C07281=1116.818,241.183,-70.393,-178.585,9.836,149.565
C07282=1116.821,240.934,-70.365,-178.587,9.834,149.565
C07283=1116.826,240.686,-70.337,-178.590,9.831,149.565
C07284=1116.829,240.473,-70.314,-178.593,9.829,149.565
C07285=1116.833,240.259,-70.290,-178.594,9.827,149.565
C07286=1116.837,240.046,-70.266,-178.597,9.825,149.565
C07287=1116.841,239.833,-70.242,-178.599,9.822,149.565
C07288=1116.844,239.620,-70.219,-178.601,9.820,149.565
C07289=1116.848,239.406,-70.195,-178.603,9.818,149.565
C07290=1116.851,239.193,-70.171,-178.605,9.816,149.565
C07291=1116.856,238.980,-70.147,-178.608,9.814,149.565
C07292=1116.860,238.732,-70.119,-178.610,9.811,149.565
C07293=1116.864,238.483,-70.092,-178.612,9.809,149.566
C07294=1116.869,238.235,-70.064,-178.615,9.806,149.566
C07295=1116.873,237.987,-70.036,-178.618,9.804,149.566
C07296=1116.877,237.738,-70.009,-178.620,9.801,149.566
C07297=1116.881,237.490,-69.981,-178.623,9.799,149.566
C07298=1116.886,237.242,-69.954,-178.626,9.796,149.566
C07299=1116.890,236.992,-69.927,-178.628,9.794,149.566
C07300=1116.894,236.744,-69.899,-178.631,9.791,149.566
C07301=1116.899,236.496,-69.872,-178.634,9.788,149.566
C07302=1116.903,236.247,-69.844,-178.637,9.785,149.566
C07303=1116.907,235.999,-69.817,-178.639,9.783,149.566
C07304=1116.912,235.751,-69.789,-178.642,9.780,149.567
C07305=1116.916,235.502,-69.761,-178.645,9.778,149.567
C07306=1116.921,235.253,-69.734,-178.648,9.775,149.567
C07307=1116.925,235.005,-69.707,-178.650,9.772,149.567
C07308=1116.930,234.757,-69.680,-178.653,9.769,149.567
C07309=1116.934,234.508,-69.652,-178.656,9.766,149.567
C07310=1116.938,234.260,-69.624,-178.659,9.764,149.567
C07311=1116.943,234.011,-69.597,-178.662,9.761,149.567
C07312=1116.946,233.762,-69.570,-178.665,9.758,149.567
C07313=1116.950,233.515,-69.543,-178.668,9.755,149.567
C07314=1116.955,233.266,-69.516,-178.671,9.753,149.568
C07315=1116.960,233.018,-69.489,-178.674,9.750,149.567
C07316=1116.964,232.768,-69.461,-178.677,9.747,149.568
C07317=1116.968,232.521,-69.433,-178.680,9.744,149.568
C07318=1116.973,232.272,-69.406,-178.682,9.741,149.568
C07319=1116.977,232.024,-69.379,-178.685,9.739,149.568
C07320=1116.981,231.775,-69.353,-178.688,9.736,149.568
C07321=1116.985,231.526,-69.325,-178.691,9.733,149.568
C07322=1116.990,231.278,-69.298,-178.694,9.730,149.568
C07323=1116.994,231.030,-69.270,-178.697,9.726,149.568
C07324=1116.999,230.781,-69.243,-178.700,9.724,149.568
C07325=1117.003,230.533,-69.217,-178.703,9.721,149.569
C07326=1117.007,230.284,-69.189,-178.706,9.718,149.569
C07327=1117.012,230.035,-69.162,-178.709,9.714,149.569
C07328=1117.016,229.787,-69.135,-178.712,9.712,149.569
C07329=1117.021,229.538,-69.108,-178.716,9.708,149.569
C07330=1117.025,229.290,-69.082,-178.719,9.705,149.569
C07331=1117.029,229.042,-69.055,-178.721,9.702,149.569
C07332=1117.034,228.793,-69.028,-178.725,9.699,149.569
C07333=1117.038,228.544,-69.000,-178.728,9.696,149.569
C07334=1117.042,228.296,-68.974,-178.730,9.693,149.569
C07335=1117.047,228.047,-68.947,-178.734,9.689,149.569
C07336=1117.051,227.799,-68.920,-178.737,9.686,149.569
C07337=1117.055,227.551,-68.893,-178.739,9.683,149.569
C07338=1117.060,227.302,-68.866,-178.742,9.681,149.569
C07339=1117.065,227.054,-68.839,-178.746,9.677,149.569
C07340=1117.068,226.840,-68.817,-178.747,9.674,149.569
C07341=1117.072,226.627,-68.793,-178.750,9.672,149.569
C07342=1117.076,226.414,-68.771,-178.753,9.669,149.569
C07343=1117.079,226.201,-68.747,-178.755,9.666,149.569
C07344=1117.083,225.987,-68.724,-178.758,9.663,149.569
C07345=1117.087,225.774,-68.702,-178.760,9.661,149.569
C07346=1117.090,225.561,-68.679,-178.762,9.658,149.569
C07347=1117.095,225.347,-68.656,-178.765,9.655,149.569
C07348=1117.099,225.099,-68.629,-178.768,9.652,149.569
C07349=1117.103,224.850,-68.602,-178.770,9.649,149.569
C07350=1117.107,224.601,-68.575,-178.773,9.646,149.569
C07351=1117.111,224.352,-68.549,-178.775,9.643,149.569
C07352=1117.116,224.104,-68.522,-178.778,9.640,149.569
C07353=1117.120,223.856,-68.496,-178.781,9.636,149.569
C07354=1117.125,223.607,-68.469,-178.784,9.633,149.569
C07355=1117.129,223.358,-68.443,-178.786,9.630,149.569
C07356=1117.134,223.110,-68.416,-178.789,9.627,149.569
C07357=1117.138,222.861,-68.389,-178.792,9.624,149.569
C07358=1117.142,222.613,-68.363,-178.794,9.621,149.569
C07359=1117.146,222.364,-68.336,-178.797,9.618,149.569
C07360=1117.151,222.115,-68.310,-178.799,9.614,149.569
C07361=1117.155,221.867,-68.284,-178.802,9.611,149.569
C07362=1117.160,221.619,-68.257,-178.804,9.608,149.569
C07363=1117.164,221.370,-68.231,-178.807,9.605,149.568
C07364=1117.169,221.121,-68.204,-178.809,9.602,149.568
C07365=1117.174,220.873,-68.178,-178.812,9.599,149.568
C07366=1117.178,220.625,-68.151,-178.814,9.595,149.568
C07367=1117.182,220.376,-68.126,-178.816,9.592,149.568
C07368=1117.187,220.127,-68.099,-178.819,9.589,149.568
C07369=1117.191,219.879,-68.072,-178.821,9.586,149.568
C07370=1117.195,219.630,-68.046,-178.824,9.583,149.568
C07371=1117.200,219.382,-68.019,-178.826,9.581,149.568
C07372=1117.204,219.133,-67.993,-178.828,9.577,149.568
C07373=1117.208,218.884,-67.968,-178.830,9.574,149.567
C07374=1117.213,218.636,-67.941,-178.833,9.571,149.567
C07375=1117.217,218.387,-67.915,-178.835,9.568,149.567
C07376=1117.222,218.139,-67.888,-178.837,9.566,149.567
C07377=1117.226,217.890,-67.862,-178.839,9.562,149.567
C07378=1117.230,217.642,-67.836,-178.842,9.559,149.567
C07379=1117.236,217.393,-67.810,-178.845,9.556,149.567
C07380=1117.240,217.144,-67.784,-178.846,9.553,149.567
C07381=1117.244,216.896,-67.757,-178.849,9.550,149.567
C07382=1117.248,216.647,-67.732,-178.851,9.547,149.566
C07383=1117.253,216.398,-67.705,-178.854,9.544,149.566
C07384=1117.257,216.150,-67.679,-178.855,9.541,149.566
C07385=1117.261,215.901,-67.653,-178.858,9.538,149.566
C07386=1117.266,215.652,-67.627,-178.859,9.536,149.566
C07387=1117.271,215.405,-67.601,-178.862,9.533,149.566
C07388=1117.275,215.156,-67.575,-178.864,9.529,149.566
C07389=1117.279,214.907,-67.549,-178.866,9.527,149.566
C07390=1117.284,214.659,-67.522,-178.869,9.524,149.566
C07391=1117.288,214.410,-67.496,-178.870,9.521,149.565
C07392=1117.292,214.161,-67.471,-178.873,9.518,149.565
C07393=1117.297,213.913,-67.445,-178.874,9.515,149.565
C07394=1117.301,213.665,-67.419,-178.877,9.512,149.565
C07395=1117.306,213.416,-67.392,-178.878,9.510,149.565
C07396=1117.309,213.202,-67.370,-178.881,9.507,149.565
C07397=1117.313,212.988,-67.349,-178.883,9.504,149.565
C07398=1117.317,212.775,-67.326,-178.885,9.502,149.565
C07399=1117.321,212.562,-67.304,-178.887,9.499,149.565
C07400=1117.325,212.348,-67.281,-178.889,9.496,149.565
C07401=1117.328,212.135,-67.259,-178.891,9.494,149.565
C07402=1117.332,211.921,-67.237,-178.894,9.491,149.565
C07403=1117.336,211.707,-67.215,-178.896,9.489,149.565
C07404=1117.340,211.459,-67.189,-178.898,9.486,149.565
C07405=1117.345,211.210,-67.164,-178.901,9.483,149.565
C07406=1117.349,210.962,-67.138,-178.903,9.480,149.565
C07407=1117.354,210.713,-67.112,-178.906,9.478,149.565
C07408=1117.359,210.464,-67.086,-178.908,9.475,149.565
C07409=1117.363,210.216,-67.061,-178.911,9.472,149.565
C07410=1117.367,209.967,-67.034,-178.914,9.469,149.565
C07411=1117.371,209.719,-67.008,-178.916,9.466,149.565
C07412=1117.376,209.471,-66.983,-178.919,9.463,149.565
C07413=1117.380,209.222,-66.957,-178.922,9.460,149.565
C07414=1117.385,208.972,-66.932,-178.925,9.457,149.565
C07415=1117.389,208.724,-66.907,-178.927,9.454,149.565
C07416=1117.394,208.475,-66.881,-178.930,9.451,149.565
C07417=1117.398,208.227,-66.855,-178.933,9.448,149.565
C07418=1117.402,207.978,-66.829,-178.936,9.445,149.565
C07419=1117.407,207.730,-66.804,-178.939,9.443,149.565
C07420=1117.411,207.481,-66.778,-178.941,9.440,149.565
C07421=1117.415,207.232,-66.753,-178.944,9.437,149.565
C07422=1117.420,206.984,-66.727,-178.947,9.434,149.565
C07423=1117.424,206.735,-66.701,-178.950,9.431,149.565
C07424=1117.429,206.486,-66.676,-178.953,9.428,149.566
C07425=1117.434,206.238,-66.651,-178.955,9.425,149.566
C07426=1117.438,205.989,-66.625,-178.958,9.422,149.566
C07427=1117.443,205.741,-66.600,-178.961,9.420,149.566
C07428=1117.447,205.492,-66.574,-178.964,9.417,149.566
C07429=1117.452,205.242,-66.549,-178.967,9.414,149.566
C07430=1117.456,204.994,-66.524,-178.969,9.411,149.566
C07431=1117.461,204.746,-66.498,-178.972,9.408,149.566
C07432=1117.465,204.497,-66.472,-178.975,9.406,149.566
C07433=1117.470,204.248,-66.448,-178.978,9.403,149.566
C07434=1117.474,203.999,-66.422,-178.981,9.400,149.566
C07435=1117.478,203.751,-66.397,-178.984,9.397,149.567
C07436=1117.483,203.503,-66.371,-178.987,9.394,149.567
C07437=1117.487,203.253,-66.346,-178.990,9.391,149.567
C07438=1117.492,203.005,-66.321,-178.993,9.388,149.567
C07439=1117.496,202.756,-66.296,-178.996,9.385,149.567
C07440=1117.501,202.508,-66.270,-178.999,9.382,149.567
C07441=1117.505,202.259,-66.245,-179.002,9.379,149.567
C07442=1117.510,202.010,-66.221,-179.004,9.376,149.567
C07443=1117.514,201.762,-66.195,-179.008,9.373,149.567
C07444=1117.519,201.512,-66.170,-179.011,9.370,149.567
C07445=1117.524,201.264,-66.144,-179.014,9.367,149.568
C07446=1117.527,201.016,-66.119,-179.016,9.364,149.568
C07447=1117.532,200.767,-66.095,-179.020,9.361,149.568
C07448=1117.536,200.518,-66.069,-179.023,9.358,149.568
C07449=1117.541,200.270,-66.045,-179.026,9.355,149.568
C07450=1117.545,200.021,-66.019,-179.028,9.352,149.568
C07451=1117.550,199.772,-65.994,-179.032,9.348,149.568
C07452=1117.554,199.558,-65.973,-179.034,9.345,149.568
C07453=1117.558,199.345,-65.952,-179.037,9.343,149.568
C07454=1117.562,199.131,-65.930,-179.040,9.341,149.568
C07455=1117.565,198.918,-65.908,-179.042,9.338,149.568
C07456=1117.569,198.704,-65.887,-179.045,9.335,149.568
C07457=1117.573,198.490,-65.866,-179.047,9.332,149.568
C07458=1117.577,198.277,-65.844,-179.050,9.330,149.568
C07459=1117.580,198.063,-65.823,-179.052,9.327,149.568
C07460=1117.586,197.814,-65.798,-179.056,9.323,149.569
C07461=1117.589,197.566,-65.773,-179.058,9.320,149.569
C07462=1117.594,197.317,-65.748,-179.062,9.317,149.569
C07463=1117.599,197.068,-65.723,-179.065,9.313,149.569
C07464=1117.603,196.820,-65.699,-179.068,9.310,149.569
C07465=1117.607,196.571,-65.674,-179.071,9.307,149.569
C07466=1117.612,196.322,-65.649,-179.074,9.303,149.569
C07467=1117.617,196.073,-65.625,-179.076,9.301,149.569
C07468=1117.620,195.825,-65.600,-179.077,9.298,149.568
C07469=1117.626,195.576,-65.575,-179.080,9.295,149.568
C07470=1117.630,195.327,-65.550,-179.081,9.292,149.568
C07471=1117.634,195.078,-65.526,-179.083,9.290,149.568
C07472=1117.640,194.830,-65.501,-179.085,9.287,149.568
C07473=1117.643,194.581,-65.476,-179.087,9.284,149.568
C07474=1117.648,194.332,-65.451,-179.089,9.282,149.568
C07475=1117.652,194.083,-65.427,-179.090,9.279,149.567
C07476=1117.657,193.835,-65.402,-179.093,9.276,149.567
C07477=1117.661,193.586,-65.378,-179.095,9.273,149.567
C07478=1117.666,193.337,-65.353,-179.097,9.270,149.567
C07479=1117.670,193.088,-65.329,-179.099,9.268,149.567
C07480=1117.675,192.840,-65.304,-179.101,9.265,149.567
C07481=1117.679,192.591,-65.279,-179.103,9.262,149.567
C07482=1117.684,192.342,-65.255,-179.105,9.260,149.567
C07483=1117.689,192.094,-65.231,-179.108,9.257,149.567
C07484=1117.693,191.845,-65.205,-179.109,9.254,149.567
C07485=1117.697,191.596,-65.181,-179.111,9.252,149.567
C07486=1117.703,191.347,-65.157,-179.114,9.249,149.567
C07487=1117.706,191.098,-65.132,-179.115,9.246,149.567
C07488=1117.711,190.850,-65.108,-179.118,9.243,149.567
C07489=1117.716,190.601,-65.084,-179.120,9.241,149.566
C07490=1117.720,190.352,-65.059,-179.122,9.238,149.566
C07491=1117.725,190.103,-65.034,-179.124,9.235,149.566
C07492=1117.729,189.855,-65.010,-179.127,9.232,149.566
C07493=1117.733,189.606,-64.986,-179.129,9.230,149.566
C07494=1117.738,189.357,-64.961,-179.131,9.226,149.566
C07495=1117.743,189.109,-64.937,-179.133,9.223,149.566
C07496=1117.748,188.860,-64.913,-179.135,9.221,149.566
C07497=1117.752,188.611,-64.888,-179.138,9.218,149.566
C07498=1117.756,188.362,-64.865,-179.140,9.216,149.566
C07499=1117.761,188.113,-64.840,-179.143,9.213,149.566
C07500=1117.766,187.865,-64.816,-179.145,9.210,149.566
C07501=1117.770,187.616,-64.792,-179.147,9.207,149.566
C07502=1117.775,187.367,-64.767,-179.150,9.204,149.566
C07503=1117.779,187.118,-64.743,-179.152,9.201,149.566
C07504=1117.783,186.870,-64.719,-179.154,9.199,149.566
C07505=1117.788,186.620,-64.694,-179.156,9.196,149.566
C07506=1117.793,186.372,-64.670,-179.159,9.193,149.566
C07507=1117.797,186.123,-64.646,-179.161,9.190,149.566
C07508=1117.801,185.910,-64.625,-179.163,9.187,149.566
C07509=1117.805,185.695,-64.604,-179.165,9.185,149.566
C07510=1117.809,185.482,-64.584,-179.167,9.183,149.566
C07511=1117.813,185.268,-64.563,-179.169,9.180,149.566
C07512=1117.817,185.055,-64.542,-179.172,9.177,149.566
C07513=1117.821,184.841,-64.522,-179.174,9.175,149.565
C07514=1117.824,184.627,-64.501,-179.176,9.173,149.566
C07515=1117.829,184.413,-64.480,-179.178,9.170,149.566
C07516=1117.833,184.165,-64.456,-179.180,9.167,149.566
C07517=1117.837,183.916,-64.432,-179.183,9.164,149.566
C07518=1117.842,183.667,-64.408,-179.185,9.161,149.565
C07519=1117.846,183.418,-64.384,-179.188,9.158,149.565
C07520=1117.850,183.170,-64.360,-179.190,9.155,149.565
C07521=1117.856,182.920,-64.336,-179.193,9.152,149.565
C07522=1117.860,182.672,-64.312,-179.195,9.149,149.565
C07523=1117.865,182.424,-64.288,-179.198,9.146,149.565
C07524=1117.869,182.175,-64.265,-179.201,9.143,149.565
C07525=1117.873,181.926,-64.240,-179.203,9.140,149.565
C07526=1117.878,181.676,-64.217,-179.206,9.137,149.565
C07527=1117.882,181.428,-64.193,-179.208,9.134,149.565
C07528=1117.888,181.179,-64.169,-179.211,9.130,149.565
C07529=1117.892,180.930,-64.145,-179.214,9.127,149.565
C07530=1117.897,180.681,-64.122,-179.216,9.124,149.565
C07531=1117.901,180.433,-64.097,-179.219,9.121,149.565
C07532=1117.906,180.184,-64.074,-179.221,9.118,149.565
C07533=1117.910,179.935,-64.050,-179.224,9.114,149.565
C07534=1117.914,179.686,-64.026,-179.227,9.111,149.565
C07535=1117.919,179.437,-64.002,-179.229,9.108,149.565
C07536=1117.923,179.188,-63.979,-179.232,9.105,149.565
C07537=1117.928,178.940,-63.955,-179.234,9.102,149.565
C07538=1117.932,178.691,-63.931,-179.236,9.099,149.565
C07539=1117.937,178.442,-63.908,-179.238,9.096,149.565
C07540=1117.942,178.193,-63.884,-179.240,9.094,149.565
C07541=1117.946,177.944,-63.861,-179.242,9.090,149.564
C07542=1117.951,177.696,-63.837,-179.245,9.087,149.564
C07543=1117.955,177.447,-63.813,-179.247,9.085,149.564
C07544=1117.960,177.198,-63.790,-179.249,9.081,149.564
C07545=1117.964,176.949,-63.766,-179.251,9.078,149.564
C07546=1117.969,176.700,-63.742,-179.253,9.076,149.564
C07547=1117.974,176.451,-63.719,-179.256,9.073,149.564
C07548=1117.979,176.202,-63.696,-179.258,9.069,149.564
C07549=1117.983,175.954,-63.672,-179.260,9.067,149.564
C07550=1117.988,175.705,-63.648,-179.262,9.064,149.564
C07551=1117.992,175.456,-63.625,-179.264,9.060,149.563
C07552=1117.997,175.207,-63.601,-179.266,9.058,149.563
C07553=1118.001,174.959,-63.578,-179.269,9.055,149.563
C07554=1118.005,174.710,-63.555,-179.271,9.051,149.563
C07555=1118.010,174.461,-63.531,-179.273,9.049,149.563
C07556=1118.015,174.212,-63.508,-179.275,9.046,149.563
C07557=1118.019,173.963,-63.484,-179.277,9.042,149.563
C07558=1118.024,173.714,-63.461,-179.279,9.040,149.563
C07559=1118.029,173.465,-63.437,-179.282,9.037,149.563
C07560=1118.033,173.216,-63.414,-179.284,9.033,149.562
C07561=1118.037,172.967,-63.391,-179.286,9.031,149.562
C07562=1118.042,172.718,-63.368,-179.288,9.028,149.562
C07563=1118.047,172.469,-63.344,-179.291,9.025,149.562
C07564=1118.050,172.256,-63.325,-179.292,9.022,149.562
C07565=1118.055,172.042,-63.304,-179.294,9.020,149.562
C07566=1118.058,171.828,-63.284,-179.296,9.017,149.562
C07567=1118.062,171.614,-63.264,-179.299,9.014,149.562
C07568=1118.066,171.400,-63.244,-179.300,9.012,149.562
C07569=1118.070,171.187,-63.224,-179.302,9.009,149.562
C07570=1118.074,170.973,-63.204,-179.304,9.007,149.562
C07571=1118.078,170.759,-63.184,-179.306,9.005,149.562
C07572=1118.082,170.510,-63.161,-179.308,9.001,149.561
C07573=1118.087,170.261,-63.138,-179.310,8.998,149.561
C07574=1118.092,170.012,-63.114,-179.313,8.995,149.561
C07575=1118.097,169.763,-63.091,-179.314,8.992,149.561
C07576=1118.101,169.515,-63.068,-179.317,8.989,149.561
C07577=1118.105,169.266,-63.045,-179.319,8.986,149.561
C07578=1118.111,169.017,-63.022,-179.321,8.983,149.561
C07579=1118.114,168.769,-62.999,-179.323,8.980,149.561
C07580=1118.119,168.520,-62.976,-179.326,8.977,149.561
C07581=1118.124,168.270,-62.952,-179.328,8.974,149.560
C07582=1118.129,168.021,-62.930,-179.330,8.971,149.560
C07583=1118.133,167.772,-62.907,-179.333,8.967,149.560
C07584=1118.138,167.523,-62.884,-179.334,8.965,149.560
C07585=1118.143,167.275,-62.861,-179.337,8.962,149.560
C07586=1118.147,167.026,-62.838,-179.339,8.958,149.560
C07587=1118.152,166.777,-62.814,-179.342,8.955,149.560
C07588=1118.156,166.528,-62.791,-179.344,8.952,149.560
C07589=1118.160,166.279,-62.769,-179.346,8.950,149.560
C07590=1118.166,166.030,-62.746,-179.348,8.946,149.559
C07591=1118.170,165.781,-62.723,-179.351,8.943,149.559
C07592=1118.174,165.533,-62.700,-179.353,8.940,149.559
C07593=1118.179,165.284,-62.677,-179.355,8.936,149.559
C07594=1118.183,165.034,-62.655,-179.358,8.933,149.559
C07595=1118.189,164.786,-62.632,-179.360,8.931,149.559
C07596=1118.193,164.537,-62.609,-179.362,8.927,149.559
C07597=1118.197,164.288,-62.585,-179.364,8.924,149.559
C07598=1118.202,164.038,-62.563,-179.367,8.921,149.559
C07599=1118.206,163.790,-62.540,-179.369,8.918,149.559
C07600=1118.212,163.541,-62.517,-179.371,8.915,149.559
C07601=1118.216,163.292,-62.495,-179.373,8.911,149.558
C07602=1118.221,163.043,-62.472,-179.376,8.908,149.558
C07603=1118.225,162.794,-62.449,-179.378,8.906,149.558
C07604=1118.230,162.545,-62.427,-179.380,8.902,149.558
C07605=1118.234,162.297,-62.404,-179.382,8.899,149.558
C07606=1118.239,162.047,-62.381,-179.385,8.896,149.558
C07607=1118.243,161.798,-62.358,-179.387,8.893,149.558
C07608=1118.248,161.550,-62.335,-179.390,8.889,149.558
C07609=1118.253,161.301,-62.313,-179.392,8.886,149.557
C07610=1118.257,161.052,-62.290,-179.394,8.883,149.557
C07611=1118.262,160.803,-62.268,-179.396,8.879,149.557
C07612=1118.266,160.554,-62.246,-179.399,8.876,149.557
C07613=1118.271,160.305,-62.223,-179.401,8.873,149.557
C07614=1118.276,160.057,-62.201,-179.403,8.870,149.557
C07615=1118.281,159.807,-62.178,-179.406,8.867,149.557
C07616=1118.285,159.558,-62.155,-179.408,8.863,149.557
C07617=1118.290,159.309,-62.133,-179.411,8.860,149.557
C07618=1118.294,159.060,-62.110,-179.413,8.856,149.556
C07619=1118.299,158.811,-62.088,-179.415,8.853,149.556
C07620=1118.304,158.551,-62.064,-179.417,8.850,149.556
C07621=1118.309,158.290,-62.041,-179.420,8.847,149.556
C07622=1118.314,158.030,-62.017,-179.422,8.843,149.556
C07623=1118.318,157.768,-61.994,-179.424,8.840,149.556
C07624=1118.323,157.520,-61.971,-179.426,8.837,149.555
C07625=1118.327,157.271,-61.949,-179.429,8.834,149.555
C07626=1118.332,157.023,-61.926,-179.431,8.830,149.555
C07627=1118.337,156.773,-61.904,-179.433,8.827,149.555
C07628=1118.341,156.524,-61.882,-179.436,8.823,149.555
C07629=1118.346,156.276,-61.860,-179.438,8.819,149.555
C07630=1118.351,156.026,-61.837,-179.441,8.816,149.555
C07631=1118.355,155.778,-61.815,-179.443,8.813,149.554
C07632=1118.360,155.528,-61.793,-179.445,8.810,149.554
C07633=1118.364,155.279,-61.770,-179.448,8.806,149.554
C07634=1118.369,155.031,-61.748,-179.450,8.803,149.554
C07635=1118.374,154.781,-61.726,-179.452,8.799,149.554
C07636=1118.378,154.533,-61.705,-179.454,8.796,149.554
C07637=1118.383,154.284,-61.681,-179.456,8.792,149.553
C07638=1118.388,154.035,-61.660,-179.459,8.789,149.553
C07639=1118.392,153.786,-61.638,-179.462,8.785,149.553
C07640=1118.397,153.536,-61.616,-179.464,8.782,149.553
C07641=1118.401,153.288,-61.594,-179.466,8.778,149.553
C07642=1118.406,153.038,-61.571,-179.468,8.775,149.553
C07643=1118.411,152.790,-61.549,-179.471,8.772,149.553
C07644=1118.415,152.541,-61.527,-179.473,8.768,149.552
C07645=1118.420,152.292,-61.505,-179.475,8.765,149.552
C07646=1118.424,152.043,-61.483,-179.478,8.761,149.552
C07647=1118.429,151.794,-61.461,-179.480,8.758,149.552
C07648=1118.434,151.544,-61.439,-179.482,8.754,149.552
C07649=1118.439,151.296,-61.417,-179.484,8.751,149.551
C07650=1118.443,151.046,-61.395,-179.486,8.747,149.551
C07651=1118.448,150.798,-61.373,-179.490,8.743,149.551
C07652=1118.453,150.548,-61.351,-179.492,8.740,149.551
C07653=1118.457,150.300,-61.330,-179.494,8.736,149.551
C07654=1118.462,150.051,-61.308,-179.496,8.733,149.550
C07655=1118.467,149.802,-61.286,-179.499,8.728,149.550
C07656=1118.471,149.553,-61.264,-179.501,8.725,149.550
C07657=1118.476,149.304,-61.242,-179.503,8.722,149.550
C07658=1118.481,149.055,-61.220,-179.505,8.718,149.550
C07659=1118.486,148.805,-61.198,-179.508,8.714,149.549
C07660=1118.490,148.557,-61.176,-179.510,8.711,149.549
C07661=1118.495,148.307,-61.154,-179.512,8.707,149.549
C07662=1118.500,148.059,-61.132,-179.514,8.704,149.549
C07663=1118.504,147.810,-61.111,-179.517,8.699,149.549
C07664=1118.509,147.560,-61.089,-179.519,8.696,149.548
C07665=1118.514,147.312,-61.068,-179.521,8.693,149.548
C07666=1118.518,147.062,-61.046,-179.524,8.689,149.548
C07667=1118.523,146.814,-61.024,-179.526,8.685,149.548
C07668=1118.530,146.397,-60.988,-179.530,8.679,149.547
C07669=1118.538,145.981,-60.952,-179.534,8.672,149.547
C07670=1118.546,145.565,-60.915,-179.538,8.666,149.547
C07671=1118.554,145.149,-60.880,-179.541,8.660,149.546
C07672=1118.558,144.935,-60.861,-179.543,8.657,149.546
C07673=1118.562,144.720,-60.843,-179.545,8.653,149.545
C07674=1118.566,144.506,-60.824,-179.546,8.651,149.545
C07675=1118.570,144.293,-60.805,-179.547,8.647,149.545
C07676=1118.574,144.078,-60.788,-179.548,8.645,149.545
C07677=1118.578,143.864,-60.768,-179.550,8.642,149.544
C07678=1118.582,143.651,-60.750,-179.551,8.639,149.544
C07679=1118.586,143.436,-60.732,-179.552,8.636,149.544
C07680=1118.591,143.187,-60.710,-179.554,8.633,149.543
C07681=1118.595,142.938,-60.689,-179.555,8.630,149.543
C07682=1118.600,142.689,-60.668,-179.558,8.626,149.543
C07683=1118.605,142.440,-60.646,-179.559,8.623,149.542
C07684=1118.609,142.191,-60.624,-179.561,8.620,149.542
C07685=1118.614,141.942,-60.603,-179.562,8.616,149.542
C07686=1118.618,141.694,-60.582,-179.564,8.613,149.541
C07687=1118.624,141.444,-60.561,-179.565,8.609,149.541
C07688=1118.628,141.195,-60.539,-179.567,8.606,149.541
C07689=1118.633,140.946,-60.518,-179.568,8.603,149.540
C07690=1118.638,140.697,-60.496,-179.570,8.599,149.540
C07691=1118.642,140.447,-60.476,-179.571,8.596,149.540
C07692=1118.647,140.199,-60.454,-179.574,8.592,149.539
C07693=1118.652,139.950,-60.432,-179.575,8.589,149.539
C07694=1118.657,139.701,-60.411,-179.577,8.586,149.539
C07695=1118.660,139.452,-60.390,-179.578,8.582,149.538
C07696=1118.665,139.203,-60.369,-179.580,8.579,149.538
C07697=1118.671,138.953,-60.348,-179.582,8.576,149.538
C07698=1118.675,138.705,-60.327,-179.583,8.573,149.537
C07699=1118.679,138.455,-60.306,-179.585,8.569,149.537
C07700=1118.684,138.206,-60.284,-179.587,8.565,149.537
C07701=1118.689,137.957,-60.263,-179.588,8.563,149.537
C07702=1118.693,137.709,-60.242,-179.590,8.559,149.536
C07703=1118.699,137.460,-60.221,-179.591,8.556,149.536
C07704=1118.703,137.210,-60.199,-179.593,8.553,149.536
C07705=1118.707,136.961,-60.178,-179.595,8.549,149.535
C07706=1118.713,136.712,-60.157,-179.596,8.546,149.535
C07707=1118.717,136.463,-60.136,-179.598,8.543,149.535
C07708=1118.722,136.214,-60.115,-179.599,8.539,149.534
C07709=1118.726,135.964,-60.094,-179.601,8.536,149.534
C07710=1118.731,135.716,-60.072,-179.603,8.532,149.534
C07711=1118.736,135.467,-60.052,-179.604,8.529,149.533
C07712=1118.741,135.218,-60.031,-179.607,8.526,149.533
C07713=1118.745,134.969,-60.011,-179.608,8.522,149.533
C07714=1118.750,134.720,-59.989,-179.610,8.519,149.533
C07715=1118.755,134.470,-59.968,-179.612,8.516,149.532
C07716=1118.759,134.221,-59.947,-179.613,8.513,149.532
C07717=1118.764,133.972,-59.926,-179.615,8.509,149.532
C07718=1118.769,133.724,-59.905,-179.617,8.506,149.531
C07719=1118.774,133.474,-59.884,-179.618,8.503,149.531
C07720=1118.779,133.225,-59.863,-179.620,8.499,149.531
C07721=1118.783,132.976,-59.843,-179.622,8.496,149.531
C07722=1118.788,132.727,-59.821,-179.623,8.493,149.530
C07723=1118.792,132.478,-59.800,-179.625,8.489,149.530
C07724=1118.797,132.228,-59.780,-179.626,8.486,149.530
C07725=1118.802,131.980,-59.759,-179.629,8.483,149.529
C07726=1118.807,131.730,-59.738,-179.630,8.479,149.529
C07727=1118.811,131.481,-59.718,-179.632,8.476,149.529
C07728=1118.815,131.267,-59.699,-179.633,8.474,149.529
C07729=1118.820,131.053,-59.681,-179.635,8.470,149.528
C07730=1118.823,130.839,-59.664,-179.637,8.467,149.528
C07731=1118.827,130.625,-59.646,-179.638,8.465,149.528
C07732=1118.831,130.411,-59.628,-179.639,8.462,149.528
C07733=1118.836,130.196,-59.610,-179.640,8.459,149.527
C07734=1118.839,129.983,-59.592,-179.642,8.456,149.527
C07735=1118.844,129.769,-59.574,-179.643,8.453,149.527
C07736=1118.849,129.520,-59.553,-179.645,8.450,149.527
C07737=1118.853,129.271,-59.533,-179.647,8.446,149.526
C07738=1118.858,129.022,-59.513,-179.648,8.443,149.526
C07739=1118.863,128.772,-59.492,-179.651,8.440,149.526
C07740=1118.867,128.523,-59.471,-179.653,8.436,149.525
C07741=1118.873,128.274,-59.450,-179.654,8.434,149.525
C07742=1118.877,128.025,-59.430,-179.656,8.430,149.525
C07743=1118.882,127.776,-59.409,-179.658,8.426,149.525
C07744=1118.887,127.527,-59.389,-179.659,8.423,149.524
C07745=1118.891,127.278,-59.368,-179.661,8.420,149.524
C07746=1118.896,127.029,-59.347,-179.663,8.416,149.524
C07747=1118.901,126.780,-59.327,-179.664,8.413,149.523
C07748=1118.905,126.531,-59.307,-179.666,8.410,149.523
C07749=1118.910,126.281,-59.285,-179.668,8.406,149.523
C07750=1118.914,126.031,-59.266,-179.669,8.403,149.523
C07751=1118.919,125.782,-59.245,-179.672,8.400,149.522
C07752=1118.925,125.534,-59.225,-179.674,8.396,149.522
C07753=1118.929,125.285,-59.204,-179.676,8.393,149.522
C07754=1118.933,125.036,-59.184,-179.677,8.390,149.522
C07755=1118.939,124.787,-59.163,-179.679,8.386,149.521
C07756=1118.943,124.538,-59.143,-179.681,8.383,149.521
C07757=1118.948,124.289,-59.122,-179.682,8.380,149.521
C07758=1118.953,124.039,-59.102,-179.684,8.377,149.521
C07759=1118.957,123.790,-59.082,-179.686,8.373,149.520
C07760=1118.962,123.541,-59.061,-179.687,8.370,149.520
C07761=1118.966,123.292,-59.041,-179.689,8.366,149.520
C07762=1118.972,123.042,-59.021,-179.692,8.363,149.519
C07763=1118.976,122.793,-59.000,-179.693,8.359,149.519
C07764=1118.981,122.544,-58.980,-179.695,8.356,149.519
C07765=1118.985,122.295,-58.959,-179.697,8.353,149.519
C07766=1118.991,122.045,-58.939,-179.699,8.349,149.518
C07767=1118.995,121.797,-58.919,-179.700,8.347,149.518
C07768=1118.999,121.548,-58.898,-179.702,8.343,149.518
C07769=1119.004,121.299,-58.878,-179.704,8.339,149.517
C07770=1119.009,121.050,-58.859,-179.706,8.336,149.517
C07771=1119.014,120.801,-58.838,-179.707,8.333,149.517
C07772=1119.019,120.552,-58.817,-179.709,8.329,149.517
C07773=1119.024,120.302,-58.798,-179.711,8.326,149.516
C07774=1119.028,120.053,-58.777,-179.713,8.322,149.516
C07775=1119.032,119.804,-58.757,-179.715,8.319,149.516
C07776=1119.037,119.555,-58.737,-179.717,8.316,149.516
C07777=1119.042,119.305,-58.716,-179.718,8.312,149.515
C07778=1119.048,119.056,-58.697,-179.720,8.309,149.515
C07779=1119.052,118.807,-58.677,-179.722,8.306,149.515
C07780=1119.057,118.558,-58.657,-179.724,8.302,149.515
C07781=1119.061,118.309,-58.637,-179.725,8.298,149.514
C07782=1119.066,118.060,-58.616,-179.727,8.295,149.514
C07783=1119.071,117.810,-58.597,-179.729,8.292,149.514
C07784=1119.075,117.597,-58.579,-179.731,8.289,149.513
C07785=1119.079,117.382,-58.563,-179.732,8.286,149.513
C07786=1119.083,117.168,-58.545,-179.734,8.283,149.513
C07787=1119.087,116.954,-58.527,-179.735,8.281,149.513
C07788=1119.092,116.740,-58.511,-179.737,8.277,149.513
C07789=1119.095,116.525,-58.493,-179.739,8.274,149.512
C07790=1119.100,116.311,-58.476,-179.740,8.271,149.512
C07791=1119.104,116.097,-58.459,-179.742,8.268,149.512
C07792=1119.108,115.848,-58.440,-179.743,8.265,149.511
C07793=1119.113,115.599,-58.419,-179.745,8.262,149.511
C07794=1119.117,115.349,-58.400,-179.747,8.258,149.511
C07795=1119.123,115.100,-58.379,-179.749,8.254,149.511
C07796=1119.128,114.851,-58.360,-179.751,8.251,149.510
C07797=1119.132,114.602,-58.339,-179.753,8.248,149.510
C07798=1119.137,114.352,-58.320,-179.755,8.244,149.510
C07799=1119.143,114.104,-58.300,-179.756,8.241,149.509
C07800=1119.147,113.855,-58.280,-179.758,8.237,149.509
C07801=1119.151,113.605,-58.261,-179.760,8.234,149.509
C07802=1119.156,113.356,-58.241,-179.762,8.230,149.509
C07803=1119.161,113.108,-58.221,-179.763,8.227,149.508
C07804=1119.165,112.858,-58.201,-179.765,8.223,149.508
C07805=1119.170,112.608,-58.182,-179.767,8.220,149.508
C07806=1119.175,112.359,-58.161,-179.769,8.216,149.507
C07807=1119.180,112.111,-58.142,-179.771,8.213,149.507
C07808=1119.185,111.861,-58.122,-179.773,8.209,149.507
C07809=1119.189,111.611,-58.103,-179.775,8.206,149.507
C07810=1119.195,111.363,-58.083,-179.776,8.203,149.506
C07811=1119.199,111.114,-58.063,-179.778,8.199,149.506
C07812=1119.204,110.864,-58.044,-179.780,8.196,149.506
C07813=1119.209,110.615,-58.024,-179.783,8.191,149.506
C07814=1119.214,110.366,-58.005,-179.785,8.188,149.505
C07815=1119.218,110.117,-57.985,-179.787,8.184,149.505
C07816=1119.223,109.868,-57.966,-179.790,8.180,149.505
C07817=1119.228,109.619,-57.946,-179.792,8.176,149.505
C07818=1119.233,109.369,-57.926,-179.794,8.173,149.504
C07819=1119.238,109.120,-57.907,-179.796,8.168,149.504
C07820=1119.243,108.871,-57.887,-179.798,8.165,149.504
C07821=1119.247,108.621,-57.868,-179.800,8.161,149.504
C07822=1119.252,108.372,-57.849,-179.803,8.157,149.503
C07823=1119.256,108.123,-57.829,-179.805,8.153,149.503
C07824=1119.261,107.874,-57.809,-179.807,8.150,149.503
C07825=1119.266,107.625,-57.790,-179.809,8.146,149.503
C07826=1119.271,107.376,-57.771,-179.811,8.142,149.502
C07827=1119.276,107.127,-57.751,-179.813,8.138,149.502
C07828=1119.281,106.877,-57.732,-179.815,8.134,149.502
C07829=1119.285,106.628,-57.713,-179.818,8.130,149.501
C07830=1119.290,106.379,-57.693,-179.820,8.127,149.501
C07831=1119.295,106.130,-57.674,-179.822,8.123,149.501
C07832=1119.300,105.881,-57.654,-179.824,8.119,149.501
C07833=1119.304,105.632,-57.635,-179.826,8.115,149.500
C07834=1119.309,105.382,-57.616,-179.828,8.111,149.500
C07835=1119.315,105.132,-57.597,-179.830,8.108,149.500
C07836=1119.319,104.883,-57.578,-179.832,8.104,149.500
C07837=1119.324,104.634,-57.559,-179.834,8.099,149.499
C07838=1119.329,104.385,-57.539,-179.836,8.096,149.499
C07839=1119.333,104.136,-57.520,-179.838,8.092,149.498
C07840=1119.338,103.922,-57.504,-179.840,8.089,149.498
C07841=1119.341,103.707,-57.487,-179.841,8.086,149.498
C07842=1119.346,103.493,-57.470,-179.843,8.082,149.498
C07843=1119.349,103.278,-57.454,-179.844,8.079,149.497
C07844=1119.354,103.064,-57.438,-179.846,8.076,149.497
C07845=1119.358,102.850,-57.422,-179.848,8.072,149.497
C07846=1119.362,102.636,-57.405,-179.849,8.069,149.496
C07847=1119.366,102.421,-57.389,-179.851,8.066,149.496
C07848=1119.371,102.172,-57.369,-179.853,8.062,149.496
C07849=1119.376,101.923,-57.350,-179.855,8.058,149.496
C07850=1119.381,101.673,-57.331,-179.857,8.054,149.495
C07851=1119.386,101.424,-57.312,-179.859,8.050,149.495
C07852=1119.390,101.175,-57.293,-179.861,8.046,149.495
C07853=1119.395,100.926,-57.274,-179.863,8.042,149.494
C07854=1119.400,100.677,-57.256,-179.865,8.039,149.494
C07855=1119.405,100.427,-57.236,-179.866,8.035,149.493
C07856=1119.409,100.179,-57.217,-179.868,8.031,149.493
C07857=1119.415,99.929,-57.199,-179.869,8.027,149.493
C07858=1119.419,99.680,-57.180,-179.872,8.024,149.492
C07859=1119.424,99.431,-57.160,-179.874,8.019,149.492
C07860=1119.429,99.181,-57.142,-179.875,8.015,149.491
C07861=1119.434,98.932,-57.123,-179.877,8.011,149.491
C07862=1119.438,98.683,-57.105,-179.879,8.008,149.491
C07863=1119.444,98.434,-57.085,-179.881,8.004,149.490
C07864=1119.448,98.184,-57.066,-179.882,8.000,149.490
C07865=1119.453,97.935,-57.048,-179.884,7.996,149.490
C07866=1119.457,97.686,-57.029,-179.885,7.992,149.489
C07867=1119.463,97.436,-57.010,-179.887,7.989,149.489
C07868=1119.468,97.188,-56.991,-179.889,7.985,149.488
C07869=1119.472,96.938,-56.973,-179.891,7.981,149.488
C07870=1119.477,96.689,-56.954,-179.892,7.977,149.488
C07871=1119.482,96.440,-56.936,-179.894,7.973,149.487
C07872=1119.487,96.190,-56.916,-179.895,7.969,149.487
C07873=1119.492,95.941,-56.898,-179.897,7.965,149.486
C07874=1119.496,95.692,-56.879,-179.899,7.961,149.486
C07875=1119.502,95.442,-56.860,-179.900,7.957,149.485
C07876=1119.506,95.194,-56.842,-179.902,7.954,149.485
C07877=1119.510,94.944,-56.823,-179.903,7.950,149.485
C07878=1119.516,94.695,-56.804,-179.905,7.946,149.484
C07879=1119.521,94.446,-56.786,-179.907,7.942,149.484
C07880=1119.525,94.196,-56.768,-179.908,7.938,149.483
C07881=1119.530,93.947,-56.748,-179.910,7.934,149.483
C07882=1119.535,93.698,-56.730,-179.911,7.930,149.482
C07883=1119.540,93.448,-56.712,-179.913,7.926,149.482
C07884=1119.545,93.199,-56.693,-179.915,7.922,149.482
C07885=1119.550,92.950,-56.675,-179.916,7.919,149.481
C07886=1119.555,92.701,-56.657,-179.918,7.915,149.481
C07887=1119.560,92.451,-56.637,-179.919,7.911,149.480
C07888=1119.564,92.202,-56.619,-179.921,7.907,149.480
C07889=1119.569,91.953,-56.601,-179.923,7.903,149.479
C07890=1119.573,91.704,-56.582,-179.924,7.899,149.479
C07891=1119.579,91.454,-56.564,-179.926,7.895,149.479
C07892=1119.584,91.205,-56.546,-179.927,7.891,149.478
C07893=1119.589,90.956,-56.528,-179.928,7.888,149.477
C07894=1119.593,90.707,-56.509,-179.930,7.884,149.477
C07895=1119.598,90.457,-56.491,-179.931,7.880,149.477
C07896=1119.603,90.242,-56.475,-179.932,7.877,149.476
C07897=1119.606,90.028,-56.459,-179.934,7.873,149.476
C07898=1119.611,89.813,-56.443,-179.935,7.870,149.475
C07899=1119.614,89.599,-56.427,-179.936,7.867,149.475
C07900=1119.619,89.385,-56.412,-179.937,7.863,149.474
C07901=1119.623,89.171,-56.396,-179.939,7.860,149.474
C07902=1119.628,88.956,-56.380,-179.940,7.857,149.474
C07903=1119.632,88.742,-56.365,-179.941,7.853,149.473
C07904=1119.637,88.493,-56.346,-179.942,7.850,149.473
C07905=1119.641,88.244,-56.328,-179.943,7.846,149.472
C07906=1119.646,87.994,-56.310,-179.945,7.842,149.472
C07907=1119.651,87.745,-56.292,-179.947,7.838,149.471
C07908=1119.656,87.496,-56.274,-179.948,7.834,149.471
C07909=1119.661,87.246,-56.255,-179.949,7.831,149.470
C07910=1119.666,86.997,-56.237,-179.950,7.827,149.470
C07911=1119.670,86.747,-56.219,-179.951,7.822,149.469
C07912=1119.675,86.498,-56.201,-179.953,7.819,149.469
C07913=1119.680,86.249,-56.183,-179.954,7.815,149.468
C07914=1119.685,86.000,-56.164,-179.955,7.811,149.468
C07915=1119.690,85.751,-56.146,-179.957,7.807,149.467
C07916=1119.695,85.502,-56.128,-179.958,7.803,149.467
C07917=1119.699,85.252,-56.110,-179.959,7.800,149.466
C07918=1119.704,85.003,-56.092,-179.960,7.796,149.466
C07919=1119.709,84.754,-56.074,-179.962,7.792,149.465
C07920=1119.714,84.504,-56.056,-179.962,7.789,149.465
C07921=1119.719,84.255,-56.038,-179.964,7.785,149.464
C07922=1119.724,84.005,-56.021,-179.965,7.780,149.464
C07923=1119.729,83.756,-56.003,-179.966,7.777,149.463
C07924=1119.733,83.506,-55.984,-179.968,7.773,149.463
C07925=1119.738,83.257,-55.966,-179.969,7.769,149.462
C07926=1119.743,83.008,-55.948,-179.970,7.766,149.462
C07927=1119.748,82.759,-55.930,-179.971,7.762,149.461
C07928=1119.753,82.510,-55.912,-179.973,7.758,149.461
C07929=1119.758,82.260,-55.894,-179.973,7.754,149.460
C07930=1119.763,82.011,-55.876,-179.975,7.750,149.460
C07931=1119.767,81.762,-55.858,-179.975,7.747,149.459
C07932=1119.772,81.513,-55.840,-179.977,7.743,149.459
C07933=1119.777,81.262,-55.823,-179.978,7.739,149.458
C07934=1119.782,81.013,-55.805,-179.979,7.736,149.457
C07935=1119.787,80.764,-55.787,-179.980,7.731,149.457
C07936=1119.792,80.515,-55.769,-179.981,7.728,149.456
C07937=1119.797,80.266,-55.751,-179.982,7.724,149.456
C07938=1119.802,80.017,-55.733,-179.983,7.721,149.455
C07939=1119.807,79.767,-55.716,-179.984,7.717,149.455
C07940=1119.812,79.518,-55.698,-179.985,7.713,149.454
C07941=1119.817,79.268,-55.680,-179.986,7.709,149.454
C07942=1119.822,79.019,-55.662,-179.987,7.706,149.453
C07943=1119.827,78.769,-55.644,-179.988,7.702,149.453
C07944=1119.831,78.521,-55.627,-179.989,7.699,149.452
C07945=1119.836,78.271,-55.609,-179.990,7.694,149.451
C07946=1119.841,78.022,-55.591,-179.991,7.691,149.451
C07947=1119.846,77.772,-55.574,-179.992,7.687,149.450
C07948=1119.851,77.523,-55.556,-179.993,7.684,149.450
C07949=1119.856,77.274,-55.538,-179.995,7.680,149.449
C07950=1119.861,77.024,-55.521,-179.995,7.676,149.449
C07951=1119.865,76.775,-55.503,-179.997,7.672,149.448
C07952=1119.869,76.561,-55.488,-179.998,7.669,149.448
C07953=1119.873,76.346,-55.472,-179.999,7.666,149.447
C07954=1119.878,76.132,-55.457,180.000,7.662,149.447
C07955=1119.882,75.917,-55.442,179.999,7.659,149.446
C07956=1119.886,75.702,-55.427,179.997,7.655,149.446
C07957=1119.891,75.488,-55.411,179.996,7.652,149.446
C07958=1119.895,75.274,-55.397,179.995,7.649,149.445
C07959=1119.899,75.059,-55.381,179.994,7.645,149.445
C07960=1119.904,74.810,-55.364,179.992,7.641,149.444
C07961=1119.909,74.560,-55.346,179.991,7.637,149.444
C07962=1119.914,74.311,-55.329,179.990,7.633,149.443
C07963=1119.918,74.062,-55.312,179.988,7.629,149.443
C07964=1119.923,73.813,-55.294,179.987,7.626,149.442
C07965=1119.928,73.563,-55.276,179.985,7.622,149.442
C07966=1119.933,73.314,-55.258,179.984,7.618,149.441
C07967=1119.938,73.064,-55.242,179.983,7.614,149.441
C07968=1119.943,72.815,-55.224,179.981,7.610,149.440
C07969=1119.948,72.566,-55.207,179.980,7.606,149.440
C07970=1119.953,72.317,-55.189,179.978,7.602,149.439
C07971=1119.958,72.067,-55.172,179.977,7.598,149.439
C07972=1119.963,71.818,-55.154,179.975,7.594,149.439
C07973=1119.967,71.568,-55.137,179.974,7.590,149.438
C07974=1119.972,71.319,-55.120,179.973,7.586,149.437
C07975=1119.977,71.070,-55.102,179.971,7.582,149.437
C07976=1119.982,70.820,-55.086,179.970,7.577,149.436
C07977=1119.987,70.571,-55.068,179.968,7.574,149.436
C07978=1119.992,70.321,-55.050,179.967,7.570,149.436
C07979=1119.997,70.073,-55.033,179.965,7.566,149.435
C07980=1120.002,69.823,-55.016,179.965,7.562,149.434
C07981=1120.007,69.573,-54.999,179.963,7.558,149.434
C07982=1120.011,69.324,-54.981,179.962,7.554,149.434
C07983=1120.017,69.075,-54.964,179.960,7.550,149.433
C07984=1120.021,68.825,-54.947,179.959,7.546,149.433
C07985=1120.026,68.576,-54.929,179.957,7.542,149.432
C07986=1120.032,68.327,-54.913,179.956,7.538,149.431
C07987=1120.036,68.077,-54.896,179.955,7.534,149.431
C07988=1120.041,67.828,-54.878,179.953,7.530,149.431
C07989=1120.046,67.579,-54.861,179.952,7.526,149.430
C07990=1120.051,67.329,-54.844,179.950,7.522,149.430
C07991=1120.055,67.079,-54.827,179.949,7.518,149.429
C07992=1120.061,66.831,-54.810,179.947,7.514,149.429
C07993=1120.066,66.581,-54.792,179.946,7.510,149.428
C07994=1120.071,66.332,-54.776,179.945,7.507,149.428
C07995=1120.076,66.082,-54.759,179.944,7.503,149.427
C07996=1120.080,65.832,-54.742,179.943,7.499,149.426
C07997=1120.086,65.584,-54.724,179.941,7.495,149.426
C07998=1120.090,65.334,-54.708,179.940,7.490,149.425
C07999=1120.095,65.085,-54.690,179.938,7.487,149.425
C08000=1120.100,64.835,-54.674,179.937,7.483,149.425
C08001=1120.105,64.586,-54.657,179.936,7.478,149.424
C08002=1120.110,64.337,-54.639,179.934,7.474,149.423
C08003=1120.114,64.088,-54.623,179.932,7.471,149.423
C08004=1120.120,63.838,-54.605,179.931,7.466,149.422
C08005=1120.124,63.588,-54.589,179.930,7.462,149.422
C08006=1120.130,63.339,-54.572,179.928,7.458,149.422
C08007=1120.134,63.090,-54.555,179.928,7.455,149.421
C08008=1120.139,62.875,-54.540,179.926,7.451,149.420
C08009=1120.143,62.661,-54.526,179.925,7.448,149.420
C08010=1120.147,62.445,-54.511,179.924,7.444,149.420
C08011=1120.151,62.232,-54.497,179.923,7.441,149.419
C08012=1120.156,62.016,-54.482,179.922,7.438,149.419
C08013=1120.160,61.803,-54.468,179.920,7.434,149.418
C08014=1120.164,61.587,-54.453,179.919,7.431,149.418
C08015=1120.168,61.373,-54.440,179.918,7.428,149.417
C08016=1120.174,61.123,-54.422,179.917,7.423,149.417
C08017=1120.178,60.874,-54.406,179.916,7.419,149.416
C08018=1120.183,60.625,-54.389,179.914,7.415,149.416
C08019=1120.188,60.375,-54.372,179.913,7.411,149.415
C08020=1120.193,60.126,-54.355,179.911,7.407,149.415
C08021=1120.198,59.877,-54.339,179.910,7.403,149.414
C08022=1120.203,59.627,-54.322,179.909,7.399,149.414
C08023=1120.208,59.378,-54.305,179.907,7.395,149.413
C08024=1120.213,59.129,-54.289,179.906,7.391,149.413
C08025=1120.218,58.879,-54.272,179.905,7.387,149.412
C08026=1120.222,58.630,-54.255,179.904,7.383,149.412
C08027=1120.228,58.381,-54.239,179.903,7.380,149.411
C08028=1120.232,58.131,-54.223,179.901,7.375,149.411
C08029=1120.238,57.882,-54.206,179.900,7.371,149.410
C08030=1120.243,57.632,-54.189,179.899,7.367,149.409
C08031=1120.247,57.383,-54.172,179.897,7.363,149.409
C08032=1120.253,57.134,-54.155,179.896,7.359,149.409
C08033=1120.257,56.884,-54.139,179.895,7.355,149.408
C08034=1120.262,56.634,-54.123,179.893,7.351,149.408
C08035=1120.267,56.385,-54.107,179.892,7.347,149.407
C08036=1120.272,56.136,-54.090,179.890,7.343,149.406
C08037=1120.278,55.887,-54.073,179.890,7.339,149.406
C08038=1120.282,55.637,-54.056,179.888,7.335,149.405
C08039=1120.287,55.387,-54.040,179.887,7.331,149.405
C08040=1120.292,55.138,-54.024,179.886,7.327,149.404
C08041=1120.297,54.888,-54.007,179.885,7.323,149.404
C08042=1120.302,54.640,-53.990,179.883,7.319,149.403
C08043=1120.307,54.390,-53.975,179.882,7.315,149.403
C08044=1120.312,54.141,-53.958,179.880,7.311,149.402
C08045=1120.317,53.891,-53.942,179.879,7.306,149.402
C08046=1120.322,53.642,-53.926,179.878,7.303,149.401
C08047=1120.327,53.392,-53.909,179.877,7.298,149.400
C08048=1120.332,53.143,-53.892,179.876,7.295,149.400
C08049=1120.337,52.893,-53.876,179.875,7.291,149.399
C08050=1120.341,52.644,-53.860,179.873,7.287,149.399
C08051=1120.347,52.395,-53.843,179.872,7.283,149.398
C08052=1120.351,52.145,-53.828,179.870,7.279,149.398
C08053=1120.356,51.896,-53.811,179.869,7.274,149.397
C08054=1120.361,51.646,-53.795,179.868,7.270,149.397
C08055=1120.366,51.397,-53.779,179.867,7.266,149.396
C08056=1120.372,51.147,-53.762,179.866,7.262,149.395
C08057=1120.377,50.898,-53.746,179.864,7.258,149.395
C08058=1120.381,50.648,-53.729,179.863,7.254,149.394
C08059=1120.387,50.399,-53.714,179.862,7.251,149.394
C08060=1120.391,50.150,-53.697,179.861,7.246,149.393
C08061=1120.397,49.900,-53.682,179.860,7.242,149.393
C08062=1120.401,49.651,-53.665,179.858,7.238,149.392
C08063=1120.407,49.401,-53.649,179.857,7.234,149.392
C08064=1120.411,49.187,-53.636,179.856,7.231,149.391
C08065=1120.415,48.972,-53.622,179.855,7.227,149.391
C08066=1120.419,48.758,-53.608,179.854,7.224,149.390
C08067=1120.424,48.543,-53.594,179.853,7.219,149.390
C08068=1120.428,48.328,-53.579,179.852,7.216,149.389
C08069=1120.432,48.114,-53.566,179.851,7.213,149.389
C08070=1120.436,47.899,-53.553,179.849,7.209,149.388
C08071=1120.440,47.684,-53.539,179.849,7.206,149.388
C08072=1120.445,47.435,-53.522,179.847,7.202,149.387
C08073=1120.450,47.185,-53.506,179.846,7.197,149.387
C08074=1120.455,46.936,-53.490,179.845,7.193,149.386
C08075=1120.460,46.687,-53.475,179.844,7.189,149.386
C08076=1120.465,46.436,-53.459,179.842,7.185,149.385
C08077=1120.470,46.188,-53.442,179.841,7.181,149.384
C08078=1120.475,45.938,-53.426,179.840,7.177,149.384
C08079=1120.481,45.688,-53.411,179.839,7.173,149.383
C08080=1120.486,45.439,-53.394,179.838,7.169,149.383
C08081=1120.490,45.189,-53.378,179.837,7.165,149.382
C08082=1120.495,44.940,-53.364,179.836,7.161,149.381
C08083=1120.499,44.691,-53.347,179.835,7.156,149.381
C08084=1120.505,44.441,-53.331,179.833,7.152,149.380
C08085=1120.510,44.192,-53.316,179.832,7.148,149.380
C08086=1120.515,43.942,-53.299,179.831,7.144,149.379
C08087=1120.520,43.693,-53.283,179.829,7.140,149.379
C08088=1120.526,43.444,-53.268,179.828,7.136,149.378
C08089=1120.530,43.193,-53.252,179.828,7.132,149.377
C08090=1120.535,42.945,-53.236,179.826,7.128,149.377
C08091=1120.540,42.696,-53.221,179.825,7.124,149.376
C08092=1120.545,42.446,-53.205,179.824,7.119,149.376
C08093=1120.550,42.196,-53.189,179.823,7.115,149.375
C08094=1120.556,41.947,-53.173,179.821,7.111,149.375
C08095=1120.559,41.698,-53.157,179.820,7.107,149.374
C08096=1120.565,41.448,-53.142,179.819,7.103,149.373
C08097=1120.570,41.199,-53.126,179.818,7.098,149.373
C08098=1120.575,40.949,-53.110,179.817,7.094,149.372
C08099=1120.580,40.699,-53.095,179.816,7.090,149.372
C08100=1120.585,40.450,-53.080,179.815,7.086,149.371
C08101=1120.590,40.200,-53.064,179.813,7.081,149.370
C08102=1120.595,39.951,-53.048,179.813,7.078,149.370
C08103=1120.600,39.702,-53.032,179.811,7.074,149.369
C08104=1120.605,39.453,-53.017,179.810,7.070,149.369
C08105=1120.610,39.203,-53.001,179.809,7.065,149.368
C08106=1120.615,38.953,-52.985,179.808,7.061,149.367
C08107=1120.620,38.704,-52.970,179.807,7.057,149.367
C08108=1120.625,38.455,-52.955,179.806,7.053,149.366
C08109=1120.630,38.205,-52.939,179.805,7.049,149.365
C08110=1120.635,37.955,-52.923,179.804,7.044,149.365
C08111=1120.640,37.706,-52.908,179.802,7.040,149.364
C08112=1120.645,37.457,-52.893,179.801,7.036,149.364
C08113=1120.650,37.207,-52.877,179.800,7.031,149.363
C08114=1120.655,36.958,-52.862,179.799,7.027,149.362
C08115=1120.660,36.708,-52.846,179.798,7.023,149.362
C08116=1120.665,36.459,-52.830,179.797,7.020,149.361
C08117=1120.670,36.209,-52.815,179.796,7.015,149.361
C08118=1120.675,35.960,-52.799,179.795,7.011,149.360
C08119=1120.680,35.710,-52.784,179.794,7.007,149.359
C08120=1120.685,35.495,-52.771,179.793,7.003,149.359
C08121=1120.689,35.280,-52.758,179.792,6.999,149.358
C08122=1120.693,35.066,-52.745,179.791,6.996,149.358
C08123=1120.698,34.851,-52.732,179.790,6.992,149.357
C08124=1120.702,34.636,-52.718,179.789,6.989,149.357
C08125=1120.706,34.421,-52.705,179.788,6.984,149.356
C08126=1120.711,34.206,-52.692,179.787,6.981,149.356
C08127=1120.715,33.991,-52.679,179.787,6.978,149.355
C08128=1120.720,33.742,-52.664,179.786,6.973,149.354
C08129=1120.725,33.493,-52.648,179.785,6.969,149.354
C08130=1120.730,33.244,-52.633,179.784,6.965,149.353
C08131=1120.735,32.994,-52.617,179.783,6.960,149.352
C08132=1120.740,32.744,-52.602,179.781,6.956,149.352
C08133=1120.745,32.495,-52.587,179.780,6.952,149.351
C08134=1120.750,32.245,-52.572,179.779,6.947,149.350
C08135=1120.755,31.996,-52.557,179.778,6.943,149.350
C08136=1120.760,31.747,-52.541,179.777,6.939,149.349
C08137=1120.765,31.497,-52.527,179.776,6.935,149.348
C08138=1120.770,31.247,-52.511,179.775,6.930,149.348
C08139=1120.775,30.998,-52.496,179.774,6.926,149.347
C08140=1120.780,30.748,-52.480,179.773,6.922,149.346
C08141=1120.785,30.499,-52.466,179.772,6.917,149.346
C08142=1120.791,30.249,-52.451,179.771,6.913,149.345
C08143=1120.795,30.000,-52.436,179.770,6.909,149.344
C08144=1120.801,29.750,-52.421,179.769,6.904,149.344
C08145=1120.805,29.501,-52.406,179.768,6.900,149.343
C08146=1120.810,29.252,-52.391,179.767,6.896,149.343
C08147=1120.816,29.002,-52.376,179.766,6.892,149.342
C08148=1120.820,28.752,-52.360,179.765,6.888,149.341
C08149=1120.825,28.503,-52.345,179.764,6.884,149.341
C08150=1120.830,28.253,-52.331,179.763,6.879,149.340
C08151=1120.836,28.004,-52.315,179.762,6.875,149.339
C08152=1120.840,27.755,-52.300,179.761,6.870,149.338
C08153=1120.845,27.505,-52.286,179.760,6.866,149.338
C08154=1120.851,27.255,-52.270,179.759,6.862,149.337
C08155=1120.856,27.006,-52.256,179.758,6.857,149.336
C08156=1120.860,26.757,-52.241,179.757,6.853,149.336
C08157=1120.866,26.507,-52.226,179.756,6.849,149.335
C08158=1120.871,26.258,-52.211,179.755,6.844,149.334
C08159=1120.876,26.008,-52.195,179.754,6.840,149.334
C08160=1120.881,25.758,-52.181,179.753,6.835,149.333
C08161=1120.886,25.509,-52.166,179.752,6.831,149.332
C08162=1120.891,25.259,-52.151,179.751,6.827,149.332
C08163=1120.896,25.010,-52.136,179.750,6.822,149.331
C08164=1120.901,24.761,-52.122,179.749,6.818,149.330
C08165=1120.907,24.510,-52.107,179.749,6.813,149.329
C08166=1120.911,24.261,-52.092,179.748,6.809,149.329
C08167=1120.916,24.012,-52.078,179.747,6.805,149.328
C08168=1120.921,23.763,-52.063,179.745,6.800,149.328
C08169=1120.926,23.513,-52.048,179.744,6.796,149.327
C08170=1120.931,23.263,-52.033,179.744,6.791,149.326
C08171=1120.936,23.014,-52.019,179.743,6.787,149.325
C08172=1120.942,22.764,-52.004,179.742,6.783,149.325
C08173=1120.946,22.515,-51.989,179.741,6.778,149.324
C08174=1120.951,22.265,-51.975,179.740,6.774,149.323
C08175=1120.956,22.016,-51.960,179.739,6.769,149.323
C08176=1120.961,21.800,-51.947,179.739,6.766,149.322
C08177=1120.965,21.586,-51.935,179.738,6.762,149.321
C08178=1120.969,21.371,-51.922,179.737,6.758,149.321
C08179=1120.973,21.156,-51.910,179.736,6.754,149.320
C08180=1120.978,20.942,-51.897,179.735,6.751,149.319
C08181=1120.983,20.727,-51.884,179.734,6.746,149.319
C08182=1120.987,20.512,-51.872,179.734,6.743,149.318
C08183=1120.992,20.297,-51.859,179.733,6.739,149.317
C08184=1120.996,20.048,-51.844,179.732,6.735,149.317
C08185=1121.001,19.798,-51.830,179.731,6.731,149.316
C08186=1121.006,19.548,-51.816,179.731,6.726,149.315
C08187=1121.011,19.298,-51.801,179.730,6.722,149.315
C08188=1121.016,19.049,-51.786,179.729,6.717,149.314
C08189=1121.022,18.799,-51.772,179.727,6.712,149.313
C08190=1121.027,18.550,-51.757,179.726,6.707,149.312
C08191=1121.032,18.301,-51.743,179.726,6.703,149.312
C08192=1121.037,18.051,-51.729,179.725,6.698,149.311
C08193=1121.042,17.802,-51.714,179.724,6.694,149.310
C08194=1121.047,17.552,-51.700,179.723,6.689,149.309
C08195=1121.052,17.302,-51.686,179.722,6.685,149.309
C08196=1121.057,17.053,-51.671,179.722,6.680,149.308
C08197=1121.062,16.803,-51.656,179.721,6.676,149.307
C08198=1121.068,16.554,-51.642,179.720,6.671,149.306
C08199=1121.073,16.305,-51.627,179.719,6.667,149.306
C08200=1121.078,16.055,-51.613,179.718,6.662,149.305
C08201=1121.082,15.805,-51.599,179.717,6.658,149.304
C08202=1121.087,15.555,-51.585,179.717,6.653,149.303
C08203=1121.093,15.306,-51.571,179.716,6.649,149.303
C08204=1121.098,15.057,-51.556,179.715,6.644,149.302
C08205=1121.103,14.807,-51.542,179.714,6.640,149.301
C08206=1121.108,14.557,-51.528,179.714,6.635,149.300
C08207=1121.113,14.308,-51.514,179.713,6.631,149.300
C08208=1121.118,14.058,-51.499,179.712,6.626,149.299
C08209=1121.123,13.809,-51.485,179.711,6.622,149.298
C08210=1121.128,13.559,-51.471,179.710,6.617,149.297
C08211=1121.133,13.309,-51.457,179.709,6.613,149.297
C08212=1121.138,13.060,-51.443,179.709,6.608,149.296
C08213=1121.144,12.811,-51.429,179.708,6.603,149.295
C08214=1121.149,12.561,-51.414,179.707,6.599,149.294
C08215=1121.154,12.311,-51.400,179.707,6.594,149.293
C08216=1121.159,12.062,-51.386,179.705,6.589,149.293
C08217=1121.164,11.813,-51.372,179.705,6.584,149.292
C08218=1121.169,11.563,-51.358,179.704,6.580,149.291
C08219=1121.174,11.313,-51.343,179.703,6.575,149.290
C08220=1121.179,11.063,-51.329,179.702,6.571,149.289
C08221=1121.185,10.814,-51.315,179.701,6.566,149.289
C08222=1121.190,10.565,-51.301,179.701,6.562,149.288
C08223=1121.194,10.315,-51.287,179.700,6.557,149.287
C08224=1121.199,10.066,-51.273,179.700,6.552,149.286
C08225=1121.204,9.817,-51.259,179.699,6.548,149.285
C08226=1121.210,9.566,-51.246,179.698,6.543,149.284
C08227=1121.214,9.317,-51.231,179.698,6.538,149.284
C08228=1121.220,9.068,-51.217,179.697,6.534,149.283
C08229=1121.225,8.818,-51.203,179.696,6.529,149.282
C08230=1121.230,8.568,-51.189,179.695,6.524,149.281
C08231=1121.236,8.319,-51.175,179.694,6.519,149.280
C08232=1121.240,8.104,-51.163,179.694,6.516,149.280
C08233=1121.244,7.889,-51.151,179.694,6.512,149.279
C08234=1121.248,7.674,-51.139,179.693,6.507,149.278
C08235=1121.253,7.459,-51.127,179.693,6.504,149.277
C08236=1121.257,7.244,-51.115,179.692,6.500,149.277
C08237=1121.261,7.029,-51.103,179.692,6.496,149.276
C08238=1121.265,6.814,-51.091,179.691,6.492,149.275
C08239=1121.270,6.599,-51.080,179.691,6.489,149.275
C08240=1121.275,6.350,-51.066,179.690,6.484,149.274
C08241=1121.280,6.100,-51.052,179.690,6.479,149.273
C08242=1121.286,5.850,-51.038,179.690,6.475,149.272
C08243=1121.291,5.601,-51.024,179.689,6.470,149.271
C08244=1121.295,5.351,-51.010,179.689,6.466,149.270
C08245=1121.301,5.102,-50.997,179.688,6.461,149.269
C08246=1121.306,4.852,-50.983,179.687,6.457,149.269
C08247=1121.311,4.602,-50.969,179.687,6.452,149.268
C08248=1121.316,4.353,-50.956,179.687,6.448,149.267
C08249=1121.321,4.103,-50.942,179.686,6.443,149.266
C08250=1121.327,3.854,-50.928,179.686,6.439,149.265
C08251=1121.332,3.604,-50.914,179.685,6.434,149.264
C08252=1121.336,3.354,-50.901,179.684,6.430,149.264
C08253=1121.342,3.105,-50.887,179.684,6.425,149.263
C08254=1121.347,2.855,-50.873,179.684,6.421,149.262
C08255=1121.352,2.606,-50.860,179.683,6.416,149.261
C08256=1121.357,2.356,-50.846,179.682,6.412,149.260
C08257=1121.362,2.106,-50.832,179.682,6.407,149.259
C08258=1121.367,1.858,-50.819,179.681,6.402,149.258
C08259=1121.372,1.607,-50.805,179.680,6.398,149.258
C08260=1121.378,1.358,-50.791,179.680,6.393,149.257
C08261=1121.383,1.108,-50.778,179.680,6.389,149.256
C08262=1121.388,0.859,-50.764,179.679,6.385,149.255
C08263=1121.393,0.609,-50.751,179.678,6.380,149.254
C08264=1121.398,0.360,-50.737,179.678,6.375,149.253
C08265=1121.403,0.110,-50.724,179.677,6.371,149.253
C08266=1121.408,-0.140,-50.710,179.676,6.366,149.252
C08267=1121.413,-0.389,-50.697,179.676,6.362,149.251
C08268=1121.418,-0.639,-50.683,179.676,6.358,149.250
C08269=1121.424,-0.889,-50.670,179.675,6.353,149.249
C08270=1121.428,-1.138,-50.656,179.674,6.349,149.249
C08271=1121.434,-1.388,-50.643,179.674,6.344,149.248
C08272=1121.438,-1.637,-50.629,179.673,6.340,149.247
C08273=1121.444,-1.887,-50.616,179.672,6.335,149.246
C08274=1121.449,-2.136,-50.601,179.672,6.330,149.245
C08275=1121.454,-2.386,-50.589,179.672,6.326,149.244
C08276=1121.459,-2.636,-50.575,179.671,6.322,149.244
C08277=1121.464,-2.885,-50.562,179.670,6.317,149.243
C08278=1121.469,-3.135,-50.548,179.670,6.312,149.242
C08279=1121.475,-3.384,-50.536,179.669,6.308,149.241
C08280=1121.479,-3.634,-50.522,179.668,6.303,149.240
C08281=1121.485,-3.883,-50.509,179.668,6.299,149.239
C08282=1121.490,-4.132,-50.495,179.667,6.294,149.239
C08283=1121.495,-4.383,-50.481,179.666,6.290,149.238
C08284=1121.501,-4.632,-50.469,179.666,6.285,149.237
C08285=1121.505,-4.882,-50.455,179.666,6.281,149.236
C08286=1121.511,-5.131,-50.442,179.665,6.277,149.235
C08287=1121.516,-5.381,-50.428,179.664,6.272,149.235
C08288=1121.521,-5.596,-50.417,179.663,6.267,149.234
C08289=1121.524,-5.811,-50.406,179.663,6.264,149.233
C08290=1121.528,-6.026,-50.394,179.663,6.260,149.232
C08291=1121.533,-6.241,-50.383,179.662,6.256,149.232
C08292=1121.537,-6.457,-50.372,179.662,6.252,149.231
C08293=1121.542,-6.671,-50.361,179.661,6.249,149.230
C08294=1121.546,-6.886,-50.349,179.660,6.244,149.230
C08295=1121.551,-7.102,-50.337,179.660,6.241,149.229
C08296=1121.556,-7.351,-50.324,179.659,6.236,149.228
C08297=1121.562,-7.601,-50.312,179.659,6.231,149.227
C08298=1121.566,-7.850,-50.298,179.658,6.227,149.227
C08299=1121.572,-8.100,-50.285,179.657,6.222,149.226
C08300=1121.577,-8.349,-50.272,179.657,6.217,149.225
C08301=1121.582,-8.599,-50.259,179.656,6.213,149.224
C08302=1121.587,-8.849,-50.246,179.655,6.208,149.223
C08303=1121.592,-9.099,-50.233,179.655,6.204,149.222
C08304=1121.597,-9.348,-50.219,179.654,6.199,149.221
C08305=1121.602,-9.597,-50.206,179.653,6.195,149.221
C08306=1121.608,-9.847,-50.193,179.653,6.190,149.220
C08307=1121.613,-10.097,-50.180,179.652,6.185,149.219
C08308=1121.618,-10.346,-50.168,179.651,6.181,149.218
C08309=1121.623,-10.596,-50.154,179.651,6.176,149.217
C08310=1121.628,-10.846,-50.142,179.650,6.171,149.217
C08311=1121.633,-11.096,-50.129,179.649,6.167,149.216
C08312=1121.638,-11.345,-50.115,179.649,6.162,149.215
C08313=1121.643,-11.594,-50.102,179.648,6.158,149.214
C08314=1121.648,-11.844,-50.089,179.647,6.153,149.214
C08315=1121.654,-12.094,-50.076,179.647,6.148,149.213
C08316=1121.659,-12.343,-50.063,179.646,6.144,149.212
C08317=1121.664,-12.592,-50.051,179.645,6.139,149.211
C08318=1121.669,-12.842,-50.037,179.645,6.135,149.210
C08319=1121.674,-13.092,-50.025,179.644,6.130,149.209
C08320=1121.680,-13.341,-50.012,179.644,6.125,149.208
C08321=1121.684,-13.591,-49.999,179.643,6.121,149.208
C08322=1121.690,-13.841,-49.986,179.642,6.116,149.207
C08323=1121.695,-14.090,-49.973,179.642,6.111,149.206
C08324=1121.700,-14.340,-49.960,179.641,6.107,149.205
C08325=1121.705,-14.589,-49.948,179.640,6.102,149.204
C08326=1121.711,-14.839,-49.934,179.640,6.098,149.204
C08327=1121.716,-15.089,-49.923,179.639,6.093,149.203
C08328=1121.721,-15.339,-49.910,179.639,6.089,149.202
C08329=1121.726,-15.588,-49.897,179.638,6.084,149.201
C08330=1121.731,-15.838,-49.884,179.638,6.079,149.200
C08331=1121.737,-16.087,-49.871,179.637,6.075,149.199
C08332=1121.741,-16.337,-49.858,179.636,6.070,149.199
C08333=1121.746,-16.587,-49.846,179.636,6.065,149.198
C08334=1121.751,-16.836,-49.833,179.635,6.061,149.197
C08335=1121.757,-17.085,-49.820,179.634,6.056,149.196
C08336=1121.762,-17.336,-49.808,179.634,6.051,149.195
C08337=1121.767,-17.586,-49.795,179.633,6.046,149.194
C08338=1121.772,-17.835,-49.782,179.632,6.041,149.193
C08339=1121.778,-18.084,-49.770,179.631,6.037,149.193
C08340=1121.783,-18.333,-49.757,179.631,6.032,149.192
C08341=1121.787,-18.584,-49.745,179.630,6.027,149.191
C08342=1121.793,-18.833,-49.732,179.630,6.023,149.190
C08343=1121.798,-19.083,-49.719,179.629,6.018,149.189
C08344=1121.803,-19.298,-49.709,179.628,6.014,149.189
C08345=1121.807,-19.513,-49.697,179.628,6.010,149.188
C08346=1121.812,-19.728,-49.687,179.627,6.006,149.187
C08347=1121.816,-19.944,-49.676,179.626,6.002,149.187
C08348=1121.821,-20.158,-49.665,179.626,5.997,149.186
C08349=1121.825,-20.373,-49.655,179.625,5.993,149.185
C08350=1121.829,-20.589,-49.644,179.625,5.989,149.184
C08351=1121.834,-20.804,-49.633,179.624,5.985,149.184
C08352=1121.840,-21.054,-49.621,179.623,5.980,149.183
C08353=1121.844,-21.304,-49.608,179.623,5.976,149.182
C08354=1121.849,-21.553,-49.595,179.622,5.971,149.181
C08355=1121.855,-21.803,-49.584,179.622,5.966,149.180
C08356=1121.860,-22.052,-49.571,179.621,5.961,149.179
C08357=1121.865,-22.302,-49.558,179.620,5.956,149.179
C08358=1121.870,-22.552,-49.546,179.619,5.952,149.178
C08359=1121.875,-22.801,-49.534,179.619,5.947,149.177
C08360=1121.881,-23.050,-49.521,179.618,5.942,149.176
C08361=1121.886,-23.300,-49.509,179.617,5.937,149.175
C08362=1121.891,-23.550,-49.496,179.617,5.932,149.174
C08363=1121.896,-23.800,-49.484,179.616,5.927,149.173
C08364=1121.901,-24.049,-49.472,179.615,5.923,149.173
C08365=1121.907,-24.299,-49.460,179.614,5.917,149.172
C08366=1121.912,-24.549,-49.447,179.614,5.912,149.171
C08367=1121.917,-24.799,-49.436,179.613,5.908,149.170
C08368=1121.922,-25.048,-49.423,179.613,5.903,149.169
C08369=1121.927,-25.297,-49.410,179.612,5.897,149.168
C08370=1121.933,-25.547,-49.398,179.611,5.893,149.167
C08371=1121.938,-25.796,-49.386,179.611,5.888,149.166
C08372=1121.943,-26.046,-49.374,179.610,5.883,149.165
C08373=1121.949,-26.296,-49.362,179.611,5.880,149.164
C08374=1121.954,-26.546,-49.349,179.612,5.875,149.163
C08375=1121.959,-26.795,-49.338,179.613,5.871,149.162
C08376=1121.964,-27.045,-49.326,179.614,5.868,149.161
C08377=1121.968,-27.295,-49.313,179.615,5.863,149.160
C08378=1121.974,-27.545,-49.301,179.615,5.859,149.159
C08379=1121.979,-27.795,-49.289,179.615,5.855,149.158
C08380=1121.984,-28.044,-49.276,179.616,5.851,149.157
C08381=1121.990,-28.294,-49.264,179.617,5.846,149.155
C08382=1121.995,-28.543,-49.252,179.617,5.842,149.154
C08383=1121.999,-28.793,-49.240,179.617,5.838,149.153
C08384=1122.005,-29.043,-49.229,179.617,5.834,149.152
C08385=1122.010,-29.292,-49.216,179.618,5.830,149.151
C08386=1122.015,-29.542,-49.204,179.618,5.826,149.150
C08387=1122.021,-29.791,-49.191,179.618,5.822,149.150
C08388=1122.026,-30.041,-49.180,179.619,5.818,149.148
C08389=1122.031,-30.291,-49.168,179.619,5.814,149.147
C08390=1122.036,-30.540,-49.156,179.619,5.810,149.147
C08391=1122.041,-30.790,-49.144,179.619,5.805,149.146
C08392=1122.046,-31.039,-49.131,179.619,5.801,149.145
C08393=1122.052,-31.289,-49.119,179.620,5.797,149.144
C08394=1122.057,-31.539,-49.107,179.619,5.792,149.143
C08395=1122.062,-31.789,-49.095,179.619,5.788,149.142
C08396=1122.067,-32.038,-49.084,179.619,5.783,149.141
C08397=1122.072,-32.288,-49.072,179.619,5.779,149.140
C08398=1122.078,-32.537,-49.059,179.618,5.774,149.139
C08399=1122.083,-32.787,-49.047,179.619,5.771,149.138
C08400=1122.087,-33.002,-49.037,179.618,5.767,149.138
C08401=1122.092,-33.217,-49.027,179.618,5.762,149.137
C08402=1122.096,-33.433,-49.016,179.617,5.759,149.136
C08403=1122.100,-33.648,-49.006,179.617,5.755,149.135
C08404=1122.106,-33.863,-48.996,179.617,5.751,149.134
C08405=1122.110,-34.078,-48.986,179.616,5.747,149.134
C08406=1122.115,-34.294,-48.975,179.616,5.743,149.133
C08407=1122.119,-34.509,-48.965,179.616,5.740,149.132
C08408=1122.124,-34.759,-48.953,179.615,5.735,149.131
C08409=1122.130,-35.009,-48.941,179.615,5.730,149.131
C08410=1122.134,-35.258,-48.930,179.614,5.726,149.130
C08411=1122.140,-35.508,-48.918,179.613,5.721,149.129
C08412=1122.145,-35.757,-48.905,179.613,5.716,149.128
C08413=1122.150,-36.007,-48.894,179.612,5.712,149.127
C08414=1122.156,-36.256,-48.882,179.611,5.706,149.126
C08415=1122.161,-36.506,-48.870,179.610,5.702,149.126
C08416=1122.166,-36.756,-48.859,179.610,5.697,149.125
C08417=1122.171,-37.006,-48.847,179.609,5.693,149.124
C08418=1122.176,-37.255,-48.835,179.608,5.687,149.123
C08419=1122.182,-37.505,-48.823,179.607,5.683,149.122
C08420=1122.186,-37.755,-48.811,179.606,5.678,149.122
C08421=1122.192,-38.005,-48.800,179.605,5.673,149.121
C08422=1122.198,-38.254,-48.788,179.604,5.668,149.120
C08423=1122.202,-38.503,-48.777,179.603,5.663,149.119
C08424=1122.208,-38.753,-48.765,179.602,5.658,149.119
C08425=1122.213,-39.003,-48.753,179.601,5.652,149.118
C08426=1122.218,-39.253,-48.742,179.600,5.648,149.117
C08427=1122.223,-39.503,-48.730,179.599,5.642,149.116
C08428=1122.228,-39.753,-48.719,179.597,5.637,149.116
C08429=1122.234,-40.002,-48.707,179.595,5.632,149.115
C08430=1122.240,-40.252,-48.695,179.594,5.626,149.114
C08431=1122.244,-40.501,-48.684,179.593,5.621,149.113
C08432=1122.250,-40.751,-48.672,179.592,5.616,149.112
C08433=1122.254,-41.001,-48.661,179.590,5.611,149.112
C08434=1122.260,-41.250,-48.649,179.589,5.605,149.111
C08435=1122.265,-41.500,-48.638,179.588,5.600,149.110
C08436=1122.271,-41.750,-48.626,179.586,5.594,149.109
C08437=1122.275,-41.999,-48.615,179.585,5.588,149.109
C08438=1122.281,-42.249,-48.603,179.583,5.583,149.108
C08439=1122.286,-42.498,-48.592,179.581,5.577,149.107
C08440=1122.291,-42.748,-48.580,179.580,5.572,149.106
C08441=1122.296,-42.998,-48.569,179.578,5.566,149.106
C08442=1122.302,-43.248,-48.558,179.578,5.561,149.105
C08443=1122.307,-43.497,-48.547,179.578,5.557,149.104
C08444=1122.313,-43.747,-48.535,179.578,5.552,149.103
C08445=1122.317,-43.997,-48.523,179.578,5.546,149.101
C08446=1122.323,-44.246,-48.512,179.579,5.542,149.100
C08447=1122.328,-44.496,-48.501,179.578,5.537,149.099
C08448=1122.333,-44.746,-48.490,179.579,5.533,149.098
C08449=1122.338,-44.996,-48.478,179.579,5.528,149.097
C08450=1122.344,-45.245,-48.467,179.579,5.523,149.096
C08451=1122.349,-45.495,-48.455,179.579,5.519,149.095
C08452=1122.354,-45.745,-48.445,179.579,5.514,149.094
C08453=1122.360,-45.994,-48.433,179.580,5.509,149.093
C08454=1122.365,-46.244,-48.422,179.580,5.505,149.092
C08455=1122.370,-46.493,-48.411,179.580,5.500,149.091
C08456=1122.374,-46.709,-48.401,179.580,5.495,149.090
C08457=1122.380,-46.925,-48.391,179.580,5.491,149.089
C08458=1122.384,-47.140,-48.381,179.580,5.488,149.088
C08459=1122.389,-47.355,-48.372,179.580,5.484,149.087
C08460=1122.393,-47.570,-48.362,179.581,5.480,149.086
C08461=1122.398,-47.785,-48.353,179.581,5.475,149.085
C08462=1122.402,-48.001,-48.344,179.581,5.471,149.084
C08463=1122.407,-48.216,-48.334,179.582,5.467,149.083
C08464=1122.411,-48.465,-48.322,179.581,5.463,149.082
C08465=1122.417,-48.716,-48.311,179.582,5.458,149.081
C08466=1122.422,-48.965,-48.300,179.582,5.453,149.080
C08467=1122.427,-49.215,-48.289,179.582,5.448,149.079
C08468=1122.433,-49.465,-48.278,179.582,5.444,149.078
C08469=1122.438,-49.714,-48.267,179.582,5.439,149.077
C08470=1122.443,-49.964,-48.256,179.583,5.435,149.076
C08471=1122.448,-50.214,-48.244,179.583,5.430,149.075
C08472=1122.454,-50.463,-48.233,179.583,5.425,149.073
C08473=1122.459,-50.713,-48.223,179.583,5.420,149.072
C08474=1122.464,-50.963,-48.211,179.583,5.416,149.071
C08475=1122.469,-51.212,-48.200,179.584,5.411,149.070
C08476=1122.474,-51.462,-48.189,179.584,5.406,149.069
C08477=1122.480,-51.711,-48.179,179.584,5.402,149.068
C08478=1122.485,-51.962,-48.167,179.584,5.397,149.067
C08479=1122.490,-52.212,-48.156,179.584,5.392,149.066
C08480=1122.496,-52.461,-48.146,179.585,5.388,149.065
C08481=1122.501,-52.711,-48.134,179.584,5.383,149.064
C08482=1122.506,-52.960,-48.123,179.585,5.378,149.063
C08483=1122.511,-53.210,-48.113,179.585,5.373,149.062
C08484=1122.516,-53.460,-48.101,179.585,5.369,149.061
C08485=1122.522,-53.710,-48.090,179.585,5.364,149.059
C08486=1122.527,-53.959,-48.079,179.585,5.359,149.058
C08487=1122.533,-54.209,-48.069,179.586,5.355,149.057
C08488=1122.537,-54.458,-48.058,179.586,5.350,149.056
C08489=1122.542,-54.709,-48.047,179.586,5.346,149.055
C08490=1122.548,-54.958,-48.036,179.586,5.341,149.054
C08491=1122.553,-55.208,-48.025,179.587,5.337,149.053
C08492=1122.559,-55.457,-48.014,179.587,5.331,149.052
C08493=1122.564,-55.707,-48.003,179.586,5.327,149.051
C08494=1122.569,-55.956,-47.993,179.587,5.322,149.050
C08495=1122.575,-56.207,-47.981,179.587,5.317,149.049
C08496=1122.579,-56.456,-47.970,179.587,5.313,149.048
C08497=1122.585,-56.706,-47.960,179.587,5.308,149.047
C08498=1122.590,-56.956,-47.949,179.588,5.304,149.045
C08499=1122.595,-57.205,-47.938,179.588,5.299,149.045
C08500=1122.600,-57.455,-47.928,179.588,5.294,149.043
C08501=1122.606,-57.705,-47.916,179.588,5.289,149.042
C08502=1122.611,-57.955,-47.906,179.588,5.285,149.041
C08503=1122.617,-58.204,-47.895,179.589,5.280,149.040
C08504=1122.622,-58.454,-47.884,179.589,5.275,149.039
C08505=1122.627,-58.704,-47.874,179.589,5.271,149.038
C08506=1122.632,-58.953,-47.863,179.589,5.266,149.037
C08507=1122.638,-59.203,-47.852,179.589,5.261,149.036
C08508=1122.643,-59.453,-47.842,179.589,5.257,149.035
C08509=1122.649,-59.702,-47.830,179.590,5.252,149.034
C08510=1122.654,-59.953,-47.820,179.590,5.248,149.033
C08511=1122.659,-60.202,-47.810,179.590,5.243,149.032
C08512=1122.664,-60.418,-47.800,179.589,5.238,149.031
C08513=1122.668,-60.633,-47.792,179.589,5.234,149.030
C08514=1122.672,-60.848,-47.782,179.588,5.229,149.029
C08515=1122.677,-61.064,-47.773,179.587,5.225,149.029
C08516=1122.682,-61.279,-47.764,179.586,5.220,149.028
C08517=1122.686,-61.495,-47.754,179.586,5.216,149.027
C08518=1122.691,-61.710,-47.745,179.585,5.211,149.026
C08519=1122.695,-61.925,-47.736,179.584,5.207,149.025
C08520=1122.700,-62.175,-47.725,179.584,5.202,149.025
C08521=1122.705,-62.425,-47.715,179.583,5.196,149.024
C08522=1122.711,-62.674,-47.705,179.582,5.191,149.023
C08523=1122.716,-62.924,-47.694,179.581,5.186,149.022
C08524=1122.721,-63.173,-47.683,179.581,5.180,149.021
C08525=1122.726,-63.423,-47.673,179.580,5.176,149.020
C08526=1122.732,-63.673,-47.662,179.580,5.170,149.019
C08527=1122.737,-63.923,-47.652,179.579,5.164,149.018
C08528=1122.742,-64.173,-47.642,179.578,5.159,149.017
C08529=1122.748,-64.422,-47.632,179.577,5.154,149.016
C08530=1122.753,-64.672,-47.620,179.577,5.149,149.015
C08531=1122.758,-64.922,-47.610,179.576,5.143,149.014
C08532=1122.763,-65.172,-47.599,179.576,5.138,149.013
C08533=1122.769,-65.421,-47.589,179.575,5.133,149.012
C08534=1122.774,-65.671,-47.579,179.575,5.128,149.011
C08535=1122.779,-65.921,-47.568,179.574,5.122,149.010
C08536=1122.785,-66.171,-47.558,179.574,5.117,149.009
C08537=1122.791,-66.420,-47.548,179.573,5.112,149.008
C08538=1122.796,-66.670,-47.537,179.573,5.107,149.007
C08539=1122.801,-66.920,-47.527,179.572,5.101,149.006
C08540=1122.806,-67.170,-47.517,179.572,5.096,149.005
C08541=1122.811,-67.419,-47.507,179.571,5.090,149.004
C08542=1122.817,-67.669,-47.497,179.571,5.085,149.003
C08543=1122.822,-67.919,-47.486,179.570,5.080,149.002
C08544=1122.827,-68.169,-47.476,179.570,5.075,149.001
C08545=1122.833,-68.418,-47.466,179.570,5.070,149.000
C08546=1122.838,-68.668,-47.456,179.569,5.064,148.999
C08547=1122.843,-68.918,-47.445,179.569,5.059,148.998
C08548=1122.848,-69.167,-47.435,179.568,5.053,148.997
C08549=1122.854,-69.417,-47.425,179.568,5.049,148.996
C08550=1122.859,-69.667,-47.415,179.567,5.043,148.995
C08551=1122.864,-69.917,-47.404,179.567,5.038,148.994
C08552=1122.870,-70.166,-47.394,179.567,5.033,148.993
C08553=1122.875,-70.416,-47.384,179.566,5.027,148.992
C08554=1122.880,-70.666,-47.374,179.566,5.022,148.991
C08555=1122.886,-70.915,-47.364,179.567,5.017,148.990
C08556=1122.891,-71.165,-47.354,179.566,5.011,148.989
C08557=1122.896,-71.416,-47.344,179.566,5.006,148.988
C08558=1122.901,-71.665,-47.334,179.565,5.001,148.987
C08559=1122.907,-71.914,-47.324,179.565,4.995,148.985
C08560=1122.912,-72.164,-47.314,179.565,4.990,148.984
C08561=1122.917,-72.414,-47.303,179.565,4.985,148.983
C08562=1122.922,-72.663,-47.294,179.564,4.979,148.982
C08563=1122.928,-72.914,-47.284,179.564,4.974,148.981
C08564=1122.934,-73.163,-47.274,179.564,4.969,148.980
C08565=1122.939,-73.413,-47.264,179.564,4.964,148.979
C08566=1122.944,-73.663,-47.254,179.564,4.958,148.978
C08567=1122.950,-73.913,-47.244,179.564,4.953,148.977
C08568=1122.954,-74.128,-47.235,179.563,4.949,148.976
C08569=1122.959,-74.343,-47.227,179.564,4.945,148.975
C08570=1122.964,-74.559,-47.218,179.563,4.940,148.974
C08571=1122.968,-74.775,-47.210,179.563,4.935,148.973
C08572=1122.973,-74.990,-47.201,179.563,4.931,148.972
C08573=1122.977,-75.205,-47.193,179.563,4.926,148.971
C08574=1122.982,-75.421,-47.184,179.564,4.922,148.970
C08575=1122.986,-75.637,-47.176,179.563,4.917,148.969
C08576=1122.992,-75.886,-47.166,179.563,4.912,148.968
C08577=1122.997,-76.136,-47.155,179.564,4.907,148.967
C08578=1123.003,-76.386,-47.147,179.563,4.901,148.966
C08579=1123.008,-76.636,-47.136,179.563,4.896,148.965
C08580=1123.012,-76.885,-47.126,179.563,4.891,148.963
C08581=1123.018,-77.135,-47.117,179.563,4.886,148.962
C08582=1123.024,-77.385,-47.107,179.563,4.881,148.961
C08583=1123.029,-77.635,-47.098,179.563,4.875,148.960
C08584=1123.035,-77.884,-47.088,179.564,4.870,148.959
C08585=1123.040,-78.134,-47.077,179.564,4.865,148.958
C08586=1123.045,-78.383,-47.068,179.564,4.860,148.956
C08587=1123.050,-78.634,-47.058,179.564,4.855,148.955
C08588=1123.056,-78.884,-47.049,179.564,4.850,148.954
C08589=1123.061,-79.133,-47.039,179.563,4.844,148.953
C08590=1123.067,-79.383,-47.029,179.563,4.839,148.952
C08591=1123.072,-79.633,-47.020,179.564,4.834,148.951
C08592=1123.078,-79.882,-47.009,179.564,4.829,148.950
C08593=1123.083,-80.132,-47.001,179.564,4.823,148.948
C08594=1123.088,-80.381,-46.990,179.564,4.818,148.947
C08595=1123.094,-80.631,-46.981,179.564,4.813,148.946
C08596=1123.099,-80.882,-46.971,179.565,4.808,148.945
C08597=1123.104,-81.131,-46.962,179.565,4.802,148.944
C08598=1123.109,-81.381,-46.952,179.566,4.798,148.942
C08599=1123.114,-81.631,-46.943,179.566,4.793,148.941
C08600=1123.120,-81.880,-46.933,179.566,4.788,148.940
C08601=1123.125,-82.130,-46.924,179.566,4.783,148.939
C08602=1123.131,-82.380,-46.914,179.566,4.777,148.938
C08603=1123.136,-82.630,-46.905,179.567,4.772,148.937
C08604=1123.142,-82.879,-46.894,179.567,4.767,148.935
C08605=1123.147,-83.129,-46.886,179.567,4.762,148.934
C08606=1123.152,-83.379,-46.875,179.567,4.757,148.933
C08607=1123.158,-83.628,-46.866,179.568,4.752,148.932
C08608=1123.163,-83.879,-46.857,179.568,4.747,148.931
C08609=1123.168,-84.128,-46.847,179.569,4.742,148.929
C08610=1123.174,-84.378,-46.838,179.569,4.737,148.928
C08611=1123.179,-84.627,-46.828,179.569,4.731,148.927
C08612=1123.184,-84.877,-46.819,179.569,4.726,148.926
C08613=1123.189,-85.127,-46.809,179.570,4.722,148.925
C08614=1123.194,-85.377,-46.800,179.570,4.717,148.923
C08615=1123.200,-85.627,-46.790,179.570,4.712,148.922
C08616=1123.205,-85.877,-46.781,179.571,4.706,148.921
C08617=1123.211,-86.127,-46.771,179.572,4.702,148.920
C08618=1123.216,-86.377,-46.762,179.572,4.697,148.918
C08619=1123.221,-86.626,-46.753,179.572,4.691,148.917
C08620=1123.227,-86.876,-46.743,179.573,4.687,148.916
C08621=1123.232,-87.126,-46.734,179.573,4.682,148.915
C08622=1123.237,-87.375,-46.725,179.574,4.676,148.913
C08623=1123.243,-87.625,-46.715,179.575,4.672,148.912
C08624=1123.248,-87.840,-46.708,179.574,4.667,148.911
C08625=1123.252,-88.056,-46.700,179.575,4.663,148.910
C08626=1123.257,-88.272,-46.691,179.575,4.659,148.909
C08627=1123.262,-88.487,-46.683,179.576,4.655,148.908
C08628=1123.266,-88.703,-46.675,179.576,4.651,148.907
C08629=1123.271,-88.918,-46.668,179.577,4.646,148.906
C08630=1123.276,-89.134,-46.659,179.577,4.642,148.905
C08631=1123.280,-89.350,-46.651,179.578,4.638,148.904
C08632=1123.285,-89.599,-46.642,179.578,4.633,148.903
C08633=1123.291,-89.849,-46.632,179.579,4.628,148.901
C08634=1123.296,-90.099,-46.623,179.579,4.623,148.900
C08635=1123.302,-90.348,-46.615,179.581,4.618,148.899
C08636=1123.307,-90.598,-46.605,179.581,4.613,148.898
C08637=1123.312,-90.848,-46.596,179.582,4.609,148.896
C08638=1123.318,-91.098,-46.587,179.582,4.604,148.895
C08639=1123.323,-91.348,-46.578,179.583,4.599,148.894
C08640=1123.328,-91.597,-46.568,179.583,4.594,148.893
C08641=1123.333,-91.847,-46.559,179.584,4.589,148.892
C08642=1123.339,-92.097,-46.550,179.584,4.584,148.890
C08643=1123.345,-92.347,-46.540,179.585,4.580,148.889
C08644=1123.350,-92.597,-46.531,179.586,4.574,148.888
C08645=1123.355,-92.847,-46.523,179.587,4.570,148.887
C08646=1123.360,-93.096,-46.513,179.587,4.566,148.885
C08647=1123.366,-93.346,-46.503,179.588,4.561,148.884
C08648=1123.371,-93.596,-46.495,179.589,4.556,148.883
C08649=1123.377,-93.845,-46.486,179.590,4.551,148.882
C08650=1123.382,-94.095,-46.477,179.590,4.546,148.880
C08651=1123.388,-94.345,-46.468,179.591,4.542,148.879
C08652=1123.393,-94.594,-46.458,179.591,4.538,148.878
C08653=1123.398,-94.844,-46.449,179.592,4.532,148.877
C08654=1123.403,-95.094,-46.440,179.592,4.527,148.876
C08655=1123.409,-95.344,-46.431,179.592,4.522,148.874
C08656=1123.414,-95.594,-46.422,179.593,4.518,148.873
C08657=1123.419,-95.844,-46.413,179.593,4.513,148.872
C08658=1123.424,-96.094,-46.404,179.593,4.507,148.871
C08659=1123.431,-96.343,-46.395,179.594,4.502,148.870
C08660=1123.436,-96.593,-46.386,179.594,4.497,148.869
C08661=1123.441,-96.843,-46.377,179.595,4.493,148.867
C08662=1123.446,-97.093,-46.368,179.595,4.488,148.866
C08663=1123.451,-97.343,-46.359,179.595,4.482,148.865
C08664=1123.457,-97.592,-46.349,179.595,4.478,148.864
C08665=1123.462,-97.842,-46.340,179.595,4.473,148.863
C08666=1123.468,-98.091,-46.332,179.596,4.468,148.862
C08667=1123.473,-98.341,-46.323,179.596,4.463,148.860
C08668=1123.478,-98.591,-46.314,179.596,4.458,148.859
C08669=1123.483,-98.841,-46.305,179.596,4.453,148.858
C08670=1123.489,-99.091,-46.295,179.597,4.448,148.857
C08671=1123.495,-99.341,-46.287,179.597,4.443,148.856
C08672=1123.500,-99.590,-46.278,179.598,4.438,148.855
C08673=1123.505,-99.840,-46.269,179.598,4.433,148.853
C08674=1123.511,-100.090,-46.261,179.598,4.428,148.852
C08675=1123.516,-100.340,-46.252,179.598,4.423,148.851
C08676=1123.521,-100.590,-46.243,179.599,4.418,148.850
C08677=1123.528,-100.839,-46.234,179.599,4.413,148.849
C08678=1123.533,-101.089,-46.225,179.599,4.408,148.848
C08679=1123.538,-101.339,-46.216,179.599,4.403,148.846
C08680=1123.543,-101.554,-46.209,179.599,4.399,148.845
C08681=1123.547,-101.770,-46.201,179.600,4.394,148.844
C08682=1123.552,-101.986,-46.194,179.600,4.390,148.843
C08683=1123.556,-102.201,-46.186,179.600,4.386,148.842
C08684=1123.561,-102.417,-46.178,179.600,4.381,148.841
C08685=1123.566,-102.633,-46.171,179.601,4.377,148.840
C08686=1123.571,-102.848,-46.163,179.601,4.373,148.839
C08687=1123.575,-103.064,-46.155,179.601,4.368,148.838
C08688=1123.580,-103.314,-46.147,179.601,4.363,148.837
C08689=1123.585,-103.564,-46.138,179.601,4.358,148.836
C08690=1123.591,-103.813,-46.130,179.602,4.353,148.835
C08691=1123.596,-104.063,-46.121,179.602,4.348,148.834
C08692=1123.602,-104.313,-46.112,179.603,4.343,148.832
C08693=1123.607,-104.563,-46.103,179.602,4.338,148.831
C08694=1123.613,-104.813,-46.095,179.603,4.333,148.830
C08695=1123.618,-105.063,-46.086,179.603,4.328,148.829
C08696=1123.623,-105.312,-46.077,179.603,4.323,148.828
C08697=1123.628,-105.562,-46.069,179.603,4.317,148.827
C08698=1123.634,-105.811,-46.060,179.603,4.312,148.825
C08699=1123.640,-106.062,-46.052,179.604,4.307,148.824
C08700=1123.645,-106.312,-46.043,179.604,4.302,148.823
C08701=1123.650,-106.561,-46.034,179.604,4.297,148.822
C08702=1123.656,-106.811,-46.025,179.604,4.292,148.821
C08703=1123.661,-107.061,-46.017,179.605,4.286,148.819
C08704=1123.666,-107.311,-46.008,179.606,4.282,148.818
C08705=1123.672,-107.560,-46.000,179.606,4.277,148.817
C08706=1123.677,-107.810,-45.991,179.605,4.272,148.816
C08707=1123.683,-108.061,-45.983,179.606,4.267,148.815
C08708=1123.688,-108.310,-45.974,179.606,4.262,148.814
C08709=1123.694,-108.560,-45.965,179.606,4.257,148.813
C08710=1123.699,-108.810,-45.957,179.606,4.251,148.811
C08711=1123.705,-109.059,-45.949,179.607,4.246,148.810
C08712=1123.710,-109.309,-45.940,179.607,4.241,148.809
C08713=1123.715,-109.559,-45.932,179.607,4.236,148.808
C08714=1123.721,-109.808,-45.924,179.607,4.231,148.807
C08715=1123.726,-110.058,-45.915,179.608,4.226,148.805
C08716=1123.731,-110.309,-45.907,179.608,4.220,148.804
C08717=1123.737,-110.558,-45.898,179.608,4.215,148.803
C08718=1123.742,-110.808,-45.889,179.608,4.210,148.802
C08719=1123.748,-111.058,-45.881,179.608,4.204,148.801
C08720=1123.753,-111.307,-45.872,179.608,4.199,148.799
C08721=1123.759,-111.558,-45.864,179.609,4.194,148.798
C08722=1123.763,-111.807,-45.856,179.609,4.189,148.797
C08723=1123.769,-112.056,-45.847,179.609,4.183,148.796
C08724=1123.774,-112.307,-45.839,179.609,4.178,148.795
C08725=1123.780,-112.556,-45.831,179.609,4.173,148.794
C08726=1123.786,-112.807,-45.822,179.609,4.168,148.792
C08727=1123.791,-113.056,-45.814,179.610,4.163,148.791
C08728=1123.796,-113.306,-45.806,179.610,4.158,148.790
C08729=1123.801,-113.556,-45.797,179.610,4.153,148.789
C08730=1123.807,-113.805,-45.790,179.610,4.147,148.788
C08731=1123.813,-114.055,-45.781,179.611,4.142,148.786
C08732=1123.818,-114.306,-45.773,179.611,4.137,148.785
C08733=1123.823,-114.555,-45.765,179.611,4.131,148.784
C08734=1123.829,-114.805,-45.756,179.611,4.126,148.783
C08735=1123.834,-115.054,-45.748,179.611,4.121,148.782
C08736=1123.839,-115.271,-45.741,179.612,4.116,148.780
C08737=1123.844,-115.486,-45.734,179.612,4.112,148.779
C08738=1123.848,-115.701,-45.727,179.612,4.107,148.779
C08739=1123.853,-115.918,-45.719,179.612,4.103,148.777
C08740=1123.858,-116.133,-45.713,179.612,4.098,148.776
C08741=1123.863,-116.349,-45.706,179.612,4.094,148.775
C08742=1123.867,-116.565,-45.698,179.613,4.089,148.774
C08743=1123.871,-116.780,-45.691,179.613,4.085,148.773
C08744=1123.877,-117.031,-45.683,179.613,4.079,148.772
C08745=1123.883,-117.280,-45.675,179.613,4.073,148.771
C08746=1123.888,-117.530,-45.666,179.613,4.068,148.770
C08747=1123.893,-117.780,-45.659,179.614,4.063,148.768
C08748=1123.899,-118.030,-45.650,179.614,4.058,148.767
C08749=1123.905,-118.279,-45.643,179.614,4.052,148.766
C08750=1123.909,-118.530,-45.635,179.614,4.047,148.765
C08751=1123.915,-118.779,-45.626,179.614,4.042,148.764
C08752=1123.921,-119.029,-45.618,179.614,4.036,148.762
C08753=1123.926,-119.279,-45.611,179.615,4.031,148.761
C08754=1123.931,-119.528,-45.602,179.614,4.025,148.760
C08755=1123.937,-119.778,-45.594,179.615,4.020,148.759
C08756=1123.942,-120.028,-45.587,179.615,4.015,148.758
C08757=1123.948,-120.278,-45.578,179.615,4.010,148.756
C08758=1123.953,-120.528,-45.570,179.615,4.004,148.755
C08759=1123.959,-120.777,-45.563,179.616,3.998,148.754
C08760=1123.964,-121.027,-45.554,179.616,3.993,148.752
C08761=1123.970,-121.277,-45.546,179.616,3.988,148.751
C08762=1123.975,-121.527,-45.539,179.616,3.982,148.750
C08763=1123.981,-121.777,-45.531,179.616,3.977,148.749
C08764=1123.986,-122.026,-45.523,179.617,3.971,148.748
C08765=1123.991,-122.276,-45.515,179.617,3.966,148.746
C08766=1123.997,-122.526,-45.507,179.617,3.960,148.745
C08767=1124.002,-122.776,-45.499,179.617,3.955,148.744
C08768=1124.008,-123.026,-45.491,179.617,3.950,148.743
C08769=1124.012,-123.276,-45.483,179.617,3.943,148.741
C08770=1124.019,-123.525,-45.475,179.618,3.938,148.740
C08771=1124.024,-123.775,-45.468,179.618,3.933,148.739
C08772=1124.029,-124.025,-45.460,179.618,3.927,148.738
C08773=1124.035,-124.275,-45.453,179.618,3.922,148.737
C08774=1124.040,-124.525,-45.444,179.618,3.917,148.735
C08775=1124.046,-124.774,-45.436,179.618,3.911,148.734
C08776=1124.051,-125.024,-45.429,179.618,3.906,148.733
C08777=1124.057,-125.274,-45.420,179.619,3.900,148.731
C08778=1124.062,-125.524,-45.413,179.619,3.894,148.730
C08779=1124.068,-125.774,-45.405,179.619,3.889,148.729
C08780=1124.073,-126.024,-45.398,179.619,3.883,148.728
C08781=1124.079,-126.273,-45.390,179.619,3.878,148.727
C08782=1124.084,-126.524,-45.382,179.619,3.873,148.725
C08783=1124.090,-126.773,-45.375,179.620,3.866,148.724
C08784=1124.095,-127.023,-45.367,179.620,3.861,148.723
C08785=1124.101,-127.273,-45.359,179.620,3.855,148.721
C08786=1124.106,-127.523,-45.352,179.620,3.850,148.720
C08787=1124.111,-127.772,-45.345,179.620,3.845,148.719
C08788=1124.117,-128.023,-45.337,179.621,3.838,148.718
C08789=1124.122,-128.272,-45.329,179.621,3.833,148.716
C08790=1124.128,-128.522,-45.322,179.621,3.827,148.715
C08791=1124.133,-128.772,-45.314,179.621,3.822,148.714
C08792=1123.710,-128.762,-45.340,179.628,3.825,148.712
C08793=1123.705,-128.513,-45.347,179.628,3.832,148.714
C08794=1123.699,-128.262,-45.355,179.628,3.837,148.715
C08795=1123.694,-128.013,-45.362,179.628,3.843,148.716
C08796=1123.688,-127.763,-45.370,179.628,3.848,148.718
C08797=1123.683,-127.513,-45.378,179.628,3.854,148.719
C08798=1123.677,-127.263,-45.385,179.627,3.860,148.720
C08799=1123.672,-127.014,-45.393,179.627,3.865,148.721
C08800=1123.666,-126.763,-45.401,179.627,3.871,148.723
C08801=1123.661,-126.514,-45.408,179.627,3.876,148.724
C08802=1123.655,-126.263,-45.416,179.627,3.882,148.725
C08803=1123.650,-126.014,-45.424,179.626,3.887,148.727
C08804=1123.644,-125.765,-45.432,179.626,3.893,148.728
C08805=1123.639,-125.514,-45.440,179.626,3.899,148.729
C08806=1123.633,-125.265,-45.447,179.626,3.904,148.730
C08807=1123.629,-125.015,-45.455,179.626,3.910,148.731
C08808=1123.623,-124.765,-45.463,179.626,3.915,148.733
C08809=1123.617,-124.515,-45.470,179.625,3.921,148.734
C08810=1123.612,-124.265,-45.479,179.625,3.927,148.735
C08811=1123.606,-124.016,-45.487,179.625,3.932,148.736
C08812=1123.601,-123.766,-45.494,179.625,3.937,148.738
C08813=1123.595,-123.516,-45.502,179.625,3.943,148.739
C08814=1123.590,-123.266,-45.510,179.625,3.948,148.740
C08815=1123.585,-123.016,-45.518,179.624,3.953,148.741
C08816=1123.579,-122.767,-45.525,179.624,3.958,148.743
C08817=1123.574,-122.517,-45.534,179.624,3.965,148.744
C08818=1123.568,-122.267,-45.541,179.624,3.970,148.745
C08819=1123.563,-122.017,-45.550,179.623,3.975,148.746
C08820=1123.557,-121.767,-45.558,179.624,3.981,148.748
C08821=1123.552,-121.517,-45.566,179.623,3.986,148.749
C08822=1123.546,-121.268,-45.573,179.623,3.992,148.750
C08823=1123.541,-121.018,-45.582,179.623,3.997,148.751
C08824=1123.536,-120.768,-45.589,179.623,4.003,148.752
C08825=1123.530,-120.518,-45.597,179.623,4.008,148.754
C08826=1123.525,-120.269,-45.606,179.622,4.013,148.755
C08827=1123.520,-120.018,-45.613,179.622,4.018,148.756
C08828=1123.514,-119.769,-45.621,179.622,4.025,148.757
C08829=1123.509,-119.519,-45.630,179.622,4.030,148.759
C08830=1123.503,-119.269,-45.637,179.621,4.035,148.760
C08831=1123.498,-119.019,-45.646,179.621,4.040,148.761
C08832=1123.492,-118.770,-45.654,179.621,4.045,148.762
C08833=1123.487,-118.519,-45.662,179.621,4.051,148.764
C08834=1123.481,-118.270,-45.669,179.621,4.056,148.765
C08835=1123.476,-118.020,-45.678,179.621,4.062,148.766
C08836=1123.470,-117.770,-45.686,179.620,4.067,148.767
C08837=1123.466,-117.521,-45.694,179.620,4.072,148.768
C08838=1123.460,-117.271,-45.702,179.620,4.078,148.770
C08839=1123.454,-117.020,-45.710,179.620,4.083,148.771
C08840=1123.448,-116.771,-45.719,179.620,4.088,148.772
C08841=1123.445,-116.555,-45.726,179.619,4.092,148.773
C08842=1123.439,-116.339,-45.733,179.619,4.098,148.774
C08843=1123.435,-116.124,-45.740,179.619,4.102,148.775
C08844=1123.430,-115.908,-45.747,179.619,4.106,148.776
C08845=1123.425,-115.692,-45.754,179.619,4.111,148.777
C08846=1123.422,-115.477,-45.762,179.618,4.115,148.778
C08847=1123.416,-115.261,-45.769,179.619,4.120,148.779
C08848=1123.411,-115.045,-45.776,179.618,4.125,148.780
C08849=1123.406,-114.795,-45.784,179.618,4.131,148.782
C08850=1123.400,-114.546,-45.792,179.618,4.136,148.783
C08851=1123.395,-114.296,-45.801,179.618,4.141,148.784
C08852=1123.390,-114.046,-45.809,179.617,4.146,148.785
C08853=1123.384,-113.797,-45.817,179.617,4.151,148.786
C08854=1123.379,-113.546,-45.825,179.617,4.156,148.788
C08855=1123.373,-113.297,-45.834,179.617,4.162,148.789
C08856=1123.368,-113.046,-45.842,179.616,4.167,148.790
C08857=1123.362,-112.797,-45.851,179.616,4.172,148.791
C08858=1123.357,-112.548,-45.859,179.616,4.177,148.792
C08859=1123.352,-112.297,-45.867,179.616,4.182,148.793
C08860=1123.346,-112.048,-45.876,179.616,4.187,148.795
C08861=1123.341,-111.798,-45.884,179.616,4.193,148.796
C08862=1123.336,-111.548,-45.893,179.616,4.198,148.797
C08863=1123.330,-111.299,-45.901,179.616,4.203,148.798
C08864=1123.324,-111.048,-45.910,179.615,4.209,148.799
C08865=1123.320,-110.799,-45.918,179.615,4.214,148.801
C08866=1123.314,-110.549,-45.926,179.615,4.219,148.802
C08867=1123.309,-110.299,-45.935,179.615,4.224,148.803
C08868=1123.304,-110.049,-45.943,179.614,4.229,148.804
C08869=1123.297,-109.799,-45.951,179.614,4.234,148.805
C08870=1123.292,-109.550,-45.960,179.614,4.240,148.807
C08871=1123.287,-109.300,-45.969,179.614,4.245,148.808
C08872=1123.281,-109.050,-45.977,179.613,4.250,148.809
C08873=1123.276,-108.800,-45.986,179.613,4.255,148.810
C08874=1123.271,-108.550,-45.995,179.613,4.260,148.811
C08875=1123.265,-108.301,-46.003,179.613,4.265,148.812
C08876=1123.259,-108.051,-46.011,179.612,4.271,148.814
C08877=1123.254,-107.801,-46.020,179.612,4.276,148.815
C08878=1123.249,-107.551,-46.029,179.612,4.281,148.816
C08879=1123.243,-107.302,-46.038,179.612,4.286,148.817
C08880=1123.238,-107.051,-46.046,179.612,4.291,148.818
C08881=1123.233,-106.801,-46.055,179.612,4.296,148.819
C08882=1123.228,-106.553,-46.063,179.611,4.300,148.821
C08883=1123.223,-106.303,-46.072,179.611,4.306,148.822
C08884=1123.217,-106.052,-46.080,179.610,4.311,148.823
C08885=1123.212,-105.802,-46.089,179.610,4.316,148.824
C08886=1123.206,-105.553,-46.097,179.610,4.321,148.825
C08887=1123.200,-105.303,-46.107,179.610,4.326,148.827
C08888=1123.195,-105.053,-46.116,179.609,4.332,148.828
C08889=1123.190,-104.803,-46.125,179.609,4.337,148.829
C08890=1123.184,-104.554,-46.132,179.609,4.342,148.830
C08891=1123.179,-104.304,-46.141,179.609,4.347,148.831
C08892=1123.173,-104.054,-46.150,179.609,4.352,148.832
C08893=1123.168,-103.804,-46.159,179.609,4.357,148.833
C08894=1123.163,-103.554,-46.168,179.608,4.361,148.835
C08895=1123.157,-103.305,-46.176,179.608,4.367,148.836
C08896=1123.152,-103.055,-46.185,179.607,4.372,148.837
C08897=1123.148,-102.839,-46.193,179.608,4.376,148.838
C08898=1123.143,-102.624,-46.200,179.607,4.381,148.839
C08899=1123.139,-102.408,-46.208,179.607,4.385,148.840
C08900=1123.134,-102.192,-46.215,179.607,4.390,148.841
C08901=1123.129,-101.976,-46.223,179.607,4.394,148.842
C08902=1123.125,-101.761,-46.231,179.606,4.398,148.843
C08903=1123.120,-101.545,-46.239,179.606,4.403,148.844
C08904=1123.115,-101.330,-46.246,179.606,4.407,148.845
C08905=1123.110,-101.080,-46.254,179.606,4.412,148.846
C08906=1123.105,-100.830,-46.263,179.605,4.417,148.848
C08907=1123.099,-100.580,-46.273,179.605,4.422,148.849
C08908=1123.093,-100.331,-46.281,179.604,4.427,148.850
C08909=1123.088,-100.081,-46.290,179.604,4.432,148.851
C08910=1123.083,-99.831,-46.299,179.604,4.437,148.852
C08911=1123.078,-99.581,-46.308,179.604,4.442,148.853
C08912=1123.072,-99.331,-46.317,179.604,4.447,148.854
C08913=1123.066,-99.082,-46.326,179.603,4.451,148.856
C08914=1123.061,-98.832,-46.335,179.603,4.456,148.857
C08915=1123.056,-98.582,-46.344,179.603,4.461,148.858
C08916=1123.050,-98.332,-46.353,179.603,4.467,148.859
C08917=1123.045,-98.082,-46.362,179.602,4.472,148.860
C08918=1123.040,-97.833,-46.371,179.602,4.477,148.862
C08919=1123.034,-97.582,-46.380,179.601,4.481,148.863
C08920=1123.028,-97.333,-46.389,179.601,4.487,148.864
C08921=1123.024,-97.084,-46.398,179.601,4.492,148.865
C08922=1123.018,-96.834,-46.407,179.601,4.497,148.866
C08923=1123.013,-96.584,-46.416,179.600,4.501,148.867
C08924=1123.007,-96.334,-46.426,179.600,4.506,148.868
C08925=1123.002,-96.084,-46.434,179.600,4.511,148.870
C08926=1122.997,-95.834,-46.443,179.600,4.516,148.871
C08927=1122.992,-95.585,-46.452,179.600,4.521,148.872
C08928=1122.986,-95.334,-46.462,179.599,4.526,148.873
C08929=1122.980,-95.085,-46.470,179.599,4.531,148.874
C08930=1122.975,-94.836,-46.480,179.598,4.536,148.876
C08931=1122.970,-94.586,-46.489,179.598,4.541,148.877
C08932=1122.964,-94.336,-46.498,179.597,4.546,148.878
C08933=1122.959,-94.086,-46.507,179.597,4.550,148.879
C08934=1122.954,-93.836,-46.516,179.596,4.555,148.880
C08935=1122.948,-93.586,-46.526,179.595,4.560,148.882
C08936=1122.943,-93.337,-46.535,179.594,4.564,148.883
C08937=1122.938,-93.087,-46.544,179.594,4.569,148.884
C08938=1122.933,-92.837,-46.553,179.593,4.574,148.885
C08939=1122.927,-92.587,-46.562,179.592,4.579,148.887
C08940=1122.922,-92.337,-46.571,179.592,4.584,148.888
C08941=1122.916,-92.089,-46.581,179.591,4.588,148.889
C08942=1122.910,-91.839,-46.590,179.591,4.593,148.890
C08943=1122.905,-91.589,-46.599,179.590,4.598,148.891
C08944=1122.900,-91.339,-46.608,179.589,4.603,148.893
C08945=1122.894,-91.089,-46.617,179.589,4.607,148.894
C08946=1122.889,-90.839,-46.627,179.588,4.613,148.895
C08947=1122.884,-90.590,-46.636,179.588,4.617,148.896
C08948=1122.878,-90.339,-46.645,179.587,4.623,148.898
C08949=1122.873,-90.090,-46.655,179.586,4.627,148.899
C08950=1122.868,-89.840,-46.664,179.586,4.632,148.900
C08951=1122.862,-89.590,-46.673,179.585,4.636,148.901
C08952=1122.857,-89.340,-46.682,179.585,4.642,148.903
C08953=1122.853,-89.125,-46.690,179.584,4.646,148.904
C08954=1122.848,-88.909,-46.698,179.584,4.650,148.905
C08955=1122.843,-88.694,-46.707,179.583,4.654,148.906
C08956=1122.839,-88.478,-46.715,179.583,4.658,148.907
C08957=1122.834,-88.263,-46.723,179.582,4.663,148.908
C08958=1122.830,-88.047,-46.731,179.582,4.667,148.909
C08959=1122.825,-87.832,-46.739,179.582,4.672,148.910
C08960=1122.820,-87.616,-46.747,179.581,4.676,148.911
C08961=1122.815,-87.366,-46.756,179.580,4.680,148.912
C08962=1122.810,-87.117,-46.766,179.580,4.686,148.914
C08963=1122.805,-86.867,-46.775,179.580,4.691,148.915
C08964=1122.799,-86.617,-46.784,179.579,4.695,148.916
C08965=1122.794,-86.367,-46.794,179.579,4.700,148.917
C08966=1122.789,-86.118,-46.803,179.579,4.705,148.918
C08967=1122.783,-85.868,-46.813,179.578,4.711,148.920
C08968=1122.778,-85.618,-46.822,179.577,4.715,148.921
C08969=1122.772,-85.368,-46.832,179.577,4.720,148.922
C08970=1122.767,-85.119,-46.841,179.577,4.726,148.923
C08971=1122.761,-84.869,-46.851,179.577,4.731,148.924
C08972=1122.756,-84.619,-46.860,179.576,4.735,148.926
C08973=1122.751,-84.370,-46.869,179.576,4.740,148.927
C08974=1122.746,-84.120,-46.879,179.575,4.746,148.928
C08975=1122.741,-83.869,-46.889,179.575,4.751,148.929
C08976=1122.735,-83.619,-46.898,179.575,4.756,148.931
C08977=1122.730,-83.370,-46.908,179.574,4.761,148.932
C08978=1122.724,-83.120,-46.917,179.574,4.766,148.933
C08979=1122.719,-82.871,-46.927,179.573,4.771,148.934
C08980=1122.714,-82.620,-46.936,179.573,4.776,148.935
C08981=1122.709,-82.371,-46.946,179.573,4.781,148.936
C08982=1122.703,-82.121,-46.955,179.573,4.786,148.938
C08983=1122.698,-81.872,-46.965,179.573,4.792,148.939
C08984=1122.692,-81.622,-46.975,179.573,4.797,148.940
C08985=1122.687,-81.372,-46.984,179.572,4.802,148.941
C08986=1122.681,-81.122,-46.994,179.572,4.807,148.943
C08987=1122.676,-80.873,-47.004,179.572,4.813,148.944
C08988=1122.671,-80.622,-47.013,179.571,4.818,148.945
C08989=1122.665,-80.373,-47.023,179.571,4.823,148.946
C08990=1122.661,-80.123,-47.033,179.571,4.828,148.947
C08991=1122.655,-79.873,-47.042,179.571,4.833,148.948
C08992=1122.650,-79.624,-47.052,179.571,4.838,148.950
C08993=1122.644,-79.374,-47.062,179.571,4.843,148.951
C08994=1122.639,-79.125,-47.071,179.570,4.849,148.952
C08995=1122.633,-78.874,-47.081,179.570,4.854,148.953
C08996=1122.628,-78.624,-47.091,179.570,4.859,148.954
C08997=1122.623,-78.375,-47.101,179.570,4.864,148.955
C08998=1122.617,-78.125,-47.110,179.570,4.869,148.956
C08999=1122.612,-77.875,-47.121,179.570,4.874,148.957
C09000=1122.607,-77.626,-47.130,179.570,4.879,148.959
C09001=1122.601,-77.376,-47.140,179.570,4.884,148.960
C09002=1122.596,-77.127,-47.149,179.570,4.890,148.961
C09003=1122.591,-76.876,-47.160,179.570,4.895,148.962
C09004=1122.585,-76.626,-47.169,179.569,4.900,148.963
C09005=1122.580,-76.377,-47.179,179.570,4.906,148.964
C09006=1122.575,-76.127,-47.189,179.570,4.911,148.966
C09007=1122.569,-75.877,-47.199,179.570,4.916,148.967
C09008=1122.564,-75.628,-47.208,179.570,4.921,148.968
C09009=1122.559,-75.413,-47.218,179.570,4.926,148.969
C09010=1122.555,-75.197,-47.226,179.570,4.930,148.970
C09011=1122.551,-74.981,-47.235,179.570,4.935,148.971
C09012=1122.545,-74.766,-47.243,179.570,4.940,148.972
C09013=1122.541,-74.551,-47.252,179.570,4.943,148.973
C09014=1122.536,-74.335,-47.260,179.570,4.948,148.974
C09015=1122.532,-74.119,-47.269,179.570,4.952,148.974
C09016=1122.527,-73.904,-47.277,179.570,4.957,148.975
C09017=1122.522,-73.654,-47.287,179.570,4.962,148.977
C09018=1122.517,-73.405,-47.297,179.571,4.968,148.978
C09019=1122.511,-73.155,-47.308,179.571,4.973,148.979
C09020=1122.505,-72.905,-47.317,179.571,4.978,148.980
C09021=1122.501,-72.655,-47.327,179.571,4.983,148.981
C09022=1122.495,-72.405,-47.337,179.571,4.989,148.982
C09023=1122.490,-72.156,-47.347,179.571,4.994,148.983
C09024=1122.484,-71.906,-47.358,179.572,4.999,148.984
C09025=1122.480,-71.656,-47.368,179.572,5.005,148.985
C09026=1122.474,-71.406,-47.377,179.572,5.010,148.986
C09027=1122.469,-71.157,-47.387,179.572,5.015,148.987
C09028=1122.463,-70.907,-47.398,179.573,5.021,148.989
C09029=1122.458,-70.657,-47.408,179.573,5.026,148.990
C09030=1122.453,-70.408,-47.418,179.573,5.031,148.991
C09031=1122.447,-70.158,-47.428,179.574,5.036,148.992
C09032=1122.442,-69.909,-47.438,179.574,5.042,148.993
C09033=1122.437,-69.658,-47.449,179.574,5.047,148.994
C09034=1122.431,-69.409,-47.459,179.575,5.052,148.995
C09035=1122.426,-69.159,-47.469,179.574,5.057,148.996
C09036=1122.421,-68.909,-47.479,179.575,5.063,148.997
C09037=1122.416,-68.660,-47.489,179.575,5.068,148.998
C09038=1122.410,-68.410,-47.500,179.576,5.073,148.999
C09039=1122.405,-68.160,-47.510,179.576,5.079,149.000
C09040=1122.400,-67.910,-47.520,179.577,5.084,149.001
C09041=1122.394,-67.661,-47.531,179.577,5.089,149.002
C09042=1122.389,-67.411,-47.541,179.577,5.094,149.003
C09043=1122.383,-67.161,-47.551,179.578,5.100,149.004
C09044=1122.378,-66.912,-47.562,179.578,5.105,149.005
C09045=1122.374,-66.662,-47.572,179.579,5.111,149.006
C09046=1122.368,-66.412,-47.582,179.580,5.115,149.007
C09047=1122.363,-66.162,-47.592,179.579,5.121,149.008
C09048=1122.357,-65.912,-47.603,179.580,5.126,149.009
C09049=1122.352,-65.663,-47.613,179.581,5.131,149.010
C09050=1122.347,-65.413,-47.624,179.582,5.136,149.011
C09051=1122.341,-65.164,-47.634,179.582,5.142,149.012
C09052=1122.336,-64.913,-47.645,179.583,5.147,149.013
C09053=1122.331,-64.664,-47.655,179.584,5.153,149.014
C09054=1122.325,-64.414,-47.665,179.584,5.157,149.015
C09055=1122.320,-64.164,-47.676,179.584,5.163,149.016
C09056=1122.315,-63.914,-47.686,179.585,5.168,149.017
C09057=1122.310,-63.665,-47.697,179.586,5.174,149.018
C09058=1122.304,-63.415,-47.708,179.586,5.179,149.019
C09059=1122.299,-63.166,-47.718,179.587,5.184,149.020
C09060=1122.294,-62.915,-47.728,179.588,5.189,149.021
C09061=1122.289,-62.667,-47.739,179.589,5.194,149.022
C09062=1122.284,-62.416,-47.750,179.590,5.200,149.022
C09063=1122.278,-62.167,-47.760,179.590,5.205,149.023
C09064=1122.273,-61.917,-47.771,179.591,5.210,149.024
C09065=1122.268,-61.701,-47.780,179.591,5.215,149.025
C09066=1122.264,-61.486,-47.789,179.592,5.219,149.026
C09067=1122.259,-61.270,-47.798,179.593,5.224,149.027
C09068=1122.255,-61.055,-47.807,179.593,5.229,149.027
C09069=1122.250,-60.840,-47.816,179.594,5.233,149.028
C09070=1122.246,-60.625,-47.826,179.595,5.238,149.029
C09071=1122.241,-60.410,-47.835,179.596,5.242,149.030
C09072=1122.236,-60.194,-47.845,179.596,5.247,149.031
C09073=1122.231,-59.944,-47.855,179.596,5.251,149.032
C09074=1122.226,-59.694,-47.865,179.596,5.256,149.033
C09075=1122.221,-59.445,-47.877,179.595,5.260,149.034
C09076=1122.215,-59.195,-47.887,179.595,5.265,149.035
C09077=1122.211,-58.946,-47.898,179.595,5.269,149.036
C09078=1122.205,-58.695,-47.909,179.595,5.274,149.037
C09079=1122.199,-58.446,-47.920,179.595,5.279,149.038
C09080=1122.195,-58.196,-47.931,179.594,5.284,149.039
C09081=1122.189,-57.946,-47.941,179.595,5.288,149.040
C09082=1122.184,-57.697,-47.952,179.594,5.293,149.041
C09083=1122.179,-57.447,-47.963,179.594,5.298,149.042
C09084=1122.173,-57.197,-47.974,179.594,5.302,149.043
C09085=1122.168,-56.948,-47.985,179.594,5.307,149.045
C09086=1122.163,-56.697,-47.995,179.594,5.312,149.046
C09087=1122.157,-56.449,-48.006,179.593,5.316,149.047
C09088=1122.152,-56.198,-48.017,179.593,5.321,149.048
C09089=1122.148,-55.949,-48.028,179.593,5.326,149.049
C09090=1122.141,-55.699,-48.039,179.593,5.330,149.050
C09091=1122.137,-55.449,-48.050,179.592,5.335,149.051
C09092=1122.131,-55.200,-48.060,179.592,5.340,149.052
C09093=1122.126,-54.950,-48.072,179.593,5.345,149.053
C09094=1122.121,-54.700,-48.082,179.592,5.349,149.054
C09095=1122.115,-54.451,-48.094,179.592,5.354,149.055
C09096=1122.110,-54.200,-48.104,179.592,5.358,149.056
C09097=1122.105,-53.951,-48.115,179.592,5.363,149.057
C09098=1122.100,-53.701,-48.126,179.591,5.367,149.059
C09099=1122.095,-53.451,-48.138,179.591,5.372,149.059
C09100=1122.089,-53.202,-48.149,179.591,5.377,149.061
C09101=1122.084,-52.952,-48.159,179.590,5.382,149.062
C09102=1122.079,-52.703,-48.170,179.591,5.386,149.063
C09103=1122.073,-52.453,-48.181,179.590,5.391,149.064
C09104=1122.069,-52.203,-48.193,179.590,5.396,149.065
C09105=1122.063,-51.953,-48.203,179.591,5.401,149.066
C09106=1122.058,-51.703,-48.215,179.590,5.405,149.067
C09107=1122.052,-51.455,-48.226,179.590,5.410,149.068
C09108=1122.047,-51.204,-48.236,179.590,5.414,149.069
C09109=1122.042,-50.954,-48.248,179.590,5.419,149.070
C09110=1122.037,-50.705,-48.259,179.589,5.424,149.071
C09111=1122.032,-50.455,-48.270,179.589,5.429,149.073
C09112=1122.026,-50.205,-48.281,179.589,5.433,149.073
C09113=1122.021,-49.956,-48.292,179.588,5.438,149.075
C09114=1122.016,-49.706,-48.303,179.588,5.443,149.076
C09115=1122.010,-49.456,-48.315,179.588,5.447,149.077
C09116=1122.005,-49.207,-48.326,179.588,5.452,149.078
C09117=1122.000,-48.957,-48.336,179.588,5.457,149.079
C09118=1121.995,-48.707,-48.348,179.588,5.461,149.080
C09119=1121.989,-48.458,-48.359,179.588,5.466,149.081
C09120=1121.984,-48.208,-48.370,179.587,5.471,149.082
C09121=1121.980,-47.993,-48.380,179.587,5.475,149.083
C09122=1121.975,-47.777,-48.390,179.587,5.479,149.084
C09123=1121.970,-47.562,-48.400,179.587,5.483,149.085
C09124=1121.966,-47.347,-48.409,179.587,5.487,149.086
